LIN {X 0,Y 204.883,Z 502.93,A -85,B 0,C 180,E1 -21530.063,E2 -21530.063} C_VEL
LIN {X 0,Y 207.726,Z 494.964,A -85,B 0,C 180,E1 -21532.899,E2 -21532.899} C_VEL
LIN {X 0,Y 210.33,Z 486.837,A -85,B 0,C 180,E1 -21535.21,E2 -21535.21} C_VEL
LIN {X 0,Y 212.639,Z 478.027,A -85,B 0,C 180,E1 -21537.271,E2 -21537.271} C_VEL
LIN {X 0,Y 215.435,Z 466.867,A -85,B 0,C 180,E1 -21539.299,E2 -21539.299} C_VEL
LIN {X 0,Y 217.848,Z 456.062,A -85,B 0,C 180,E1 -21540.809,E2 -21540.809} C_VEL
LIN {X 0,Y 219.818,Z 444.103,A -85,B 0,C 180,E1 -21542.111,E2 -21542.111} C_VEL
LIN {X 0,Y 221.525,Z 430.516,A -85,B 0,C 180,E1 -21543.135,E2 -21543.135} C_VEL
LIN {X 0,Y 222.579,Z 417.478,A -85,B 0,C 180,E1 -21543.751,E2 -21543.751} C_VEL
LIN {X 0,Y 224.876,Z 365.159,A -85,B 0,C 180,E1 -21545.36,E2 -21545.36} C_VEL
LIN {X 0,Y 218.22,Z 351.727,A -85,B 0,C 180,E1 -21547.162,E2 -21547.162} C_VEL
LIN {X 0,Y 211.105,Z 339.207,A -85,B 0,C 180,E1 -21549.189,E2 -21549.189} C_VEL
LIN {X 0,Y 204.724,Z 329.151,A -85,B 0,C 180,E1 -21551.13,E2 -21551.13} C_VEL
LIN {X 0,Y 202.531,Z 325.685,A -85,B 0,C 180,E1 -21551.84,E2 -21551.84} C_VEL
LIN {X 0,Y 200.323,Z 322.897,A -85,B 0,C 180,E1 -21552.544,E2 -21552.544} C_VEL
LIN {X 0,Y 199.618,Z 320.611,A -85,B 0,C 180,E1 -21552.884,E2 -21552.884} C_VEL
LIN {X 0,Y 199.586,Z 320.596,A -85,B 0,C 180,E1 -21558.006,E2 -21558.006} C_VEL
LIN {X 0,Y 199.617,Z 320.622,A -85,B 0,C 180,E1 -21560.768,E2 -21560.768} C_VEL
LIN {X 0,Y 199.619,Z 320.62,A -85,B 0,C 180,E1 -21565.714,E2 -21565.714} C_VEL
LIN {X 0,Y 199.699,Z 320.598,A -85,B 0,C 180,E1 -21568.137,E2 -21568.137} C_VEL
LIN {X 0,Y 199.782,Z 320.599,A -85,B 0,C 180,E1 -21573.034,E2 -21573.034} C_VEL
LIN {X 0,Y 206.99,Z 349.218,A -85,B 0,C 180,E1 -21575.078,E2 -21575.078} C_VEL
LIN {X 0,Y 203.484,Z 423.442,A -85,B 0,C 180,E1 -21579.706,E2 -21579.706} C_VEL
LIN {X 0,Y 202.574,Z 437.8,A -85,B 0,C 180,E1 -21581.019,E2 -21581.019} C_VEL
LIN {X 0,Y 201.78,Z 450.031,A -85,B 0,C 180,E1 -21582.518,E2 -21582.518} C_VEL
LIN {X 0,Y 201.022,Z 459.956,A -85,B 0,C 180,E1 -21584.019,E2 -21584.019} C_VEL
LIN {X 0,Y 200.03,Z 472.119,A -85,B 0,C 180,E1 -21586.281,E2 -21586.281} C_VEL
LIN {X 0,Y 199.173,Z 483.028,A -85,B 0,C 180,E1 -21588.809,E2 -21588.809} C_VEL
LIN {X 0,Y 198.588,Z 492.082,A -85,B 0,C 180,E1 -21591.349,E2 -21591.349} C_VEL
LIN {X 0,Y 198.092,Z 499.573,A -85,B 0,C 180,E1 -21593.89,E2 -21593.89} C_VEL
LIN {X 0,Y 197.871,Z 507.068,A -85,B 0,C 180,E1 -21596.946,E2 -21596.946} C_VEL
LIN {X 0,Y 197.683,Z 513.047,A -85,B 0,C 180,E1 -21600,E2 -21600} C_VEL
LIN {X 0,Y 197.864,Z 517.861,A -85,B 0,C 180,E1 -21603.054,E2 -21603.054} C_VEL
LIN {X 0,Y 198.329,Z 521.612,A -85,B 0,C 180,E1 -21606.102,E2 -21606.102} C_VEL
LIN {X 0,Y 199.664,Z 525.148,A -85,B 0,C 180,E1 -21610.137,E2 -21610.137} C_VEL
LIN {X 0,Y 202.176,Z 527.196,A -85,B 0,C 180,E1 -21614.083,E2 -21614.083} C_VEL
LIN {X 0,Y 205.529,Z 527.784,A -85,B 0,C 180,E1 -21617.924,E2 -21617.924} C_VEL
LIN {X 0,Y 210.067,Z 526.862,A -85,B 0,C 180,E1 -21621.593,E2 -21621.593} C_VEL
LIN {X 0,Y 215.556,Z 524.507,A -85,B 0,C 180,E1 -21625.078,E2 -21625.078} C_VEL
LIN {X 0,Y 221.972,Z 520.613,A -85,B 0,C 180,E1 -21628.355,E2 -21628.355} C_VEL
LIN {X 0,Y 227.936,Z 516.178,A -85,B 0,C 180,E1 -21630.852,E2 -21630.852} C_VEL
LIN {X 0,Y 230.413,Z 513.934,A -85,B 0,C 180,E1 -21632.07,E2 -21632.07} C_VEL
LIN {X 0,Y 235.965,Z 507.455,A -85,B 0,C 180,E1 -21635.911,E2 -21635.911} C_VEL
LIN {X 0,Y 238.533,Z 504.702,A -85,B 0,C 180,E1 -21636.994,E2 -21636.994} C_VEL
LIN {X 0,Y 239.576,Z 503.651,A -85,B 0,C 180,E1 -21637.301,E2 -21637.301} C_VEL
LIN {X 0,Y 246.733,Z 495.901,A -85,B 0,C 180,E1 -21639.118,E2 -21639.118} C_VEL
LIN {X 0,Y 253.535,Z 487.509,A -85,B 0,C 180,E1 -21640.649,E2 -21640.649} C_VEL
LIN {X 0,Y 260.762,Z 477.305,A -85,B 0,C 180,E1 -21642.1,E2 -21642.1} C_VEL
LIN {X 0,Y 267.508,Z 466.194,A -85,B 0,C 180,E1 -21643.343,E2 -21643.343} C_VEL
LIN {X 0,Y 273.686,Z 454.125,A -85,B 0,C 180,E1 -21644.356,E2 -21644.356} C_VEL
LIN {X 0,Y 273.26,Z 455.121,A -85,B 0,C 180,E1 -21644.754,E2 -21644.754} C_VEL
LIN {X 0,Y 266.867,Z 467.844,A -85,B 0,C 180,E1 -21645.596,E2 -21645.596} C_VEL
LIN {X 0,Y 259.241,Z 480.574,A -85,B 0,C 180,E1 -21646.747,E2 -21646.747} C_VEL
LIN {X 0,Y 253.403,Z 489.105,A -85,B 0,C 180,E1 -21647.733,E2 -21647.733} C_VEL
LIN {X 0,Y 246.637,Z 497.975,A -85,B 0,C 180,E1 -21649.049,E2 -21649.049} C_VEL
LIN {X 0,Y 238.874,Z 507.03,A -85,B 0,C 180,E1 -21650.759,E2 -21650.759} C_VEL
LIN {X 0,Y 230.486,Z 515.708,A -85,B 0,C 180,E1 -21652.969,E2 -21652.969} C_VEL
LIN {X 0,Y 222.797,Z 522.767,A -85,B 0,C 180,E1 -21655.401,E2 -21655.401} C_VEL
LIN {X 0,Y 216.779,Z 527.728,A -85,B 0,C 180,E1 -21657.659,E2 -21657.659} C_VEL
LIN {X 0,Y 209.493,Z 532.953,A -85,B 0,C 180,E1 -21660.891,E2 -21660.891} C_VEL
LIN {X 0,Y 204.769,Z 535.863,A -85,B 0,C 180,E1 -21663.499,E2 -21663.499} C_VEL
LIN {X 0,Y 199.666,Z 538.52,A -85,B 0,C 180,E1 -21667.218,E2 -21667.218} C_VEL
LIN {X 0,Y 195.58,Z 539.845,A -85,B 0,C 180,E1 -21671.129,E2 -21671.129} C_VEL
LIN {X 0,Y 192.79,Z 539.808,A -85,B 0,C 180,E1 -21675.214,E2 -21675.214} C_VEL
LIN {X 0,Y 191.317,Z 538.398,A -85,B 0,C 180,E1 -21679.414,E2 -21679.414} C_VEL
LIN {X 0,Y 191.037,Z 537.758,A -85,B 0,C 180,E1 -21680.869,E2 -21680.869} C_VEL
LIN {X 0,Y 190.528,Z 539.752,A -85,B 0,C 180,E1 -21683.645,E2 -21683.645} C_VEL
LIN {X 0,Y 190.385,Z 540.768,A -85,B 0,C 180,E1 -21685.764,E2 -21685.764} C_VEL
LIN {X 0,Y 190.403,Z 541.392,A -85,B 0,C 180,E1 -21687.883,E2 -21687.883} C_VEL
LIN {X 0,Y 190.598,Z 541.618,A -85,B 0,C 180,E1 -21689.998,E2 -21689.998} C_VEL
LIN {X 0,Y 190.41,Z 541.379,A -85,B 0,C 180,E1 -21692.113,E2 -21692.113} C_VEL
LIN {X 0,Y 190.302,Z 540.701,A -85,B 0,C 180,E1 -21694.341,E2 -21694.341} C_VEL
LIN {X 0,Y 190.306,Z 539.712,A -85,B 0,C 180,E1 -21696.359,E2 -21696.359} C_VEL
LIN {X 0,Y 190.479,Z 538.255,A -85,B 0,C 180,E1 -21698.485,E2 -21698.485} C_VEL
LIN {X 0,Y 191.094,Z 535.243,A -85,B 0,C 180,E1 -21701.668,E2 -21701.668} C_VEL
LIN {X 0,Y 192.189,Z 531.169,A -85,B 0,C 180,E1 -21704.829,E2 -21704.829} C_VEL
LIN {X 0,Y 194.299,Z 524.907,A -85,B 0,C 180,E1 -21708.449,E2 -21708.449} C_VEL
LIN {X 0,Y 196.303,Z 519.321,A -85,B 0,C 180,E1 -21710.976,E2 -21710.976} C_VEL
LIN {X 0,Y 198.955,Z 511.125,A -85,B 0,C 180,E1 -21713.966,E2 -21713.966} C_VEL
LIN {X 0,Y 201.69,Z 502.727,A -85,B 0,C 180,E1 -21716.375,E2 -21716.375} C_VEL
LIN {X 0,Y 204.869,Z 492.34,A -85,B 0,C 180,E1 -21718.701,E2 -21718.701} C_VEL
LIN {X 0,Y 207.651,Z 482.066,A -85,B 0,C 180,E1 -21720.507,E2 -21720.507} C_VEL
LIN {X 0,Y 210.277,Z 470.801,A -85,B 0,C 180,E1 -21722.042,E2 -21722.042} C_VEL
LIN {X 0,Y 212.675,Z 457.931,A -85,B 0,C 180,E1 -21723.322,E2 -21723.322} C_VEL
LIN {X 0,Y 214.527,Z 445.105,A -85,B 0,C 180,E1 -21724.193,E2 -21724.193} C_VEL
LIN {X 0,Y 215.524,Z 431.944,A -85,B 0,C 180,E1 -21724.76,E2 -21724.76} C_VEL
LIN {X 0,Y 217.316,Z 391.03,A -85,B 0,C 180,E1 -21726.05,E2 -21726.05} C_VEL
LIN {X 0,Y 214.641,Z 363.738,A -85,B 0,C 180,E1 -21727.683,E2 -21727.683} C_VEL
LIN {X 0,Y 210.098,Z 349.908,A -85,B 0,C 180,E1 -21729.23,E2 -21729.23} C_VEL
LIN {X 0,Y 204.593,Z 340.582,A -85,B 0,C 180,E1 -21730.911,E2 -21730.911} C_VEL
LIN {X 0,Y 200.055,Z 333.574,A -85,B 0,C 180,E1 -21732.368,E2 -21732.368} C_VEL
LIN {X 0,Y 197.462,Z 329.773,A -85,B 0,C 180,E1 -21733.238,E2 -21733.238} C_VEL
LIN {X 0,Y 195.165,Z 326.199,A -85,B 0,C 180,E1 -21734.048,E2 -21734.048} C_VEL
LIN {X 0,Y 193.201,Z 323.758,A -85,B 0,C 180,E1 -21734.734,E2 -21734.734} C_VEL
LIN {X 0,Y 192.549,Z 321.496,A -85,B 0,C 180,E1 -21735.102,E2 -21735.102} C_VEL
LIN {X 0,Y 192.499,Z 321.494,A -85,B 0,C 180,E1 -21740.054,E2 -21740.054} C_VEL
LIN {X 0,Y 192.551,Z 321.489,A -85,B 0,C 180,E1 -21744.268,E2 -21744.268} C_VEL
LIN {X 0,Y 192.598,Z 321.492,A -85,B 0,C 180,E1 -21747.06,E2 -21747.06} C_VEL
LIN {X 0,Y 192.612,Z 321.493,A -85,B 0,C 180,E1 -21751.683,E2 -21751.683} C_VEL
LIN {X 0,Y 192.655,Z 321.486,A -85,B 0,C 180,E1 -21756.342,E2 -21756.342} C_VEL
LIN {X 0,Y 192.687,Z 321.438,A -85,B 0,C 180,E1 -21761.491,E2 -21761.491} C_VEL
LIN {X 0,Y 192.731,Z 321.453,A -85,B 0,C 180,E1 -21765.211,E2 -21765.211} C_VEL
LIN {X 0,Y 192.938,Z 321.445,A -85,B 0,C 180,E1 -21769.566,E2 -21769.566} C_VEL
LIN {X 0,Y 192.956,Z 321.393,A -85,B 0,C 180,E1 -21773.727,E2 -21773.727} C_VEL
LIN {X 0,Y 193.222,Z 321.399,A -85,B 0,C 180,E1 -21777.916,E2 -21777.916} C_VEL
LIN {X 0,Y 193.404,Z 321.391,A -85,B 0,C 180,E1 -21780,E2 -21780} C_VEL
LIN {X 0,Y 192.924,Z 321.441,A -85,B 0,C 180,E1 -21784.178,E2 -21784.178} C_VEL
LIN {X 0,Y 193.016,Z 321.434,A -85,B 0,C 180,E1 -21788.375,E2 -21788.375} C_VEL
LIN {X 0,Y 192.784,Z 321.471,A -85,B 0,C 180,E1 -21792.635,E2 -21792.635} C_VEL
LIN {X 0,Y 192.712,Z 321.454,A -85,B 0,C 180,E1 -21796.963,E2 -21796.963} C_VEL
LIN {X 0,Y 192.602,Z 321.493,A -85,B 0,C 180,E1 -21801.401,E2 -21801.401} C_VEL
LIN {X 0,Y 192.633,Z 321.47,A -85,B 0,C 180,E1 -21804.209,E2 -21804.209} C_VEL
LIN {X 0,Y 192.596,Z 321.495,A -85,B 0,C 180,E1 -21808.867,E2 -21808.867} C_VEL
LIN {X 0,Y 192.589,Z 321.482,A -85,B 0,C 180,E1 -21813.188,E2 -21813.188} C_VEL
LIN {X 0,Y 192.545,Z 321.485,A -85,B 0,C 180,E1 -21818.354,E2 -21818.354} C_VEL
LIN {X 0,Y 192.484,Z 321.496,A -85,B 0,C 180,E1 -21823.097,E2 -21823.097} C_VEL
LIN {X 0,Y 192.549,Z 321.515,A -85,B 0,C 180,E1 -21825.4,E2 -21825.4} C_VEL
LIN {X 0,Y 193.375,Z 324.086,A -85,B 0,C 180,E1 -21825.774,E2 -21825.774} C_VEL
LIN {X 0,Y 195.707,Z 326.993,A -85,B 0,C 180,E1 -21826.585,E2 -21826.585} C_VEL
LIN {X 0,Y 197.792,Z 330.187,A -85,B 0,C 180,E1 -21827.314,E2 -21827.314} C_VEL
LIN {X 0,Y 203.771,Z 339.212,A -85,B 0,C 180,E1 -21829.272,E2 -21829.272} C_VEL
LIN {X 0,Y 210.873,Z 351.252,A -85,B 0,C 180,E1 -21831.445,E2 -21831.445} C_VEL
LIN {X 0,Y 217.687,Z 364.631,A -85,B 0,C 180,E1 -21833.415,E2 -21833.415} C_VEL
LIN {X 0,Y 218.98,Z 367.37,A -85,B 0,C 180,E1 -21833.778,E2 -21833.778} C_VEL
LIN {X 0,Y 216.238,Z 422.514,A -85,B 0,C 180,E1 -21835.528,E2 -21835.528} C_VEL
LIN {X 0,Y 215.03,Z 435.02,A -85,B 0,C 180,E1 -21836.249,E2 -21836.249} C_VEL
LIN {X 0,Y 213.234,Z 447.586,A -85,B 0,C 180,E1 -21837.339,E2 -21837.339} C_VEL
LIN {X 0,Y 211.136,Z 458.838,A -85,B 0,C 180,E1 -21838.663,E2 -21838.663} C_VEL
LIN {X 0,Y 208.673,Z 469.175,A -85,B 0,C 180,E1 -21840.216,E2 -21840.216} C_VEL
LIN {X 0,Y 206.125,Z 478.927,A -85,B 0,C 180,E1 -21842.1,E2 -21842.1} C_VEL
LIN {X 0,Y 203.422,Z 488.432,A -85,B 0,C 180,E1 -21844.43,E2 -21844.43} C_VEL
LIN {X 0,Y 200.224,Z 497.77,A -85,B 0,C 180,E1 -21847.29,E2 -21847.29} C_VEL
LIN {X 0,Y 197.517,Z 505.216,A -85,B 0,C 180,E1 -21850.246,E2 -21850.246} C_VEL
LIN {X 0,Y 195.288,Z 511.189,A -85,B 0,C 180,E1 -21853.27,E2 -21853.27} C_VEL
LIN {X 0,Y 193.48,Z 515.906,A -85,B 0,C 180,E1 -21856.345,E2 -21856.345} C_VEL
LIN {X 0,Y 192.195,Z 519.505,A -85,B 0,C 180,E1 -21859.467,E2 -21859.467} C_VEL
LIN {X 0,Y 191.243,Z 522.257,A -85,B 0,C 180,E1 -21862.852,E2 -21862.852} C_VEL
LIN {X 0,Y 190.77,Z 523.755,A -85,B 0,C 180,E1 -21865.777,E2 -21865.777} C_VEL
LIN {X 0,Y 190.523,Z 524.593,A -85,B 0,C 180,E1 -21870.002,E2 -21870.002} C_VEL
LIN {X 0,Y 190.573,Z 524.396,A -85,B 0,C 180,E1 -21872.116,E2 -21872.116} C_VEL
LIN {X 0,Y 190.77,Z 523.809,A -85,B 0,C 180,E1 -21874.228,E2 -21874.228} C_VEL
LIN {X 0,Y 191.565,Z 521.476,A -85,B 0,C 180,E1 -21878.441,E2 -21878.441} C_VEL
LIN {X 0,Y 192.512,Z 518.607,A -85,B 0,C 180,E1 -21881.585,E2 -21881.585} C_VEL
LIN {X 0,Y 193.961,Z 514.699,A -85,B 0,C 180,E1 -21884.695,E2 -21884.695} C_VEL
LIN {X 0,Y 195.918,Z 509.63,A -85,B 0,C 180,E1 -21887.755,E2 -21887.755} C_VEL
LIN {X 0,Y 198.239,Z 503.242,A -85,B 0,C 180,E1 -21890.766,E2 -21890.766} C_VEL
LIN {X 0,Y 201.218,Z 495.274,A -85,B 0,C 180,E1 -21893.684,E2 -21893.684} C_VEL
LIN {X 0,Y 203.728,Z 487.809,A -85,B 0,C 180,E1 -21895.877,E2 -21895.877} C_VEL
LIN {X 0,Y 206.372,Z 478.331,A -85,B 0,C 180,E1 -21898.172,E2 -21898.172} C_VEL
LIN {X 0,Y 209.302,Z 467.166,A -85,B 0,C 180,E1 -21900.245,E2 -21900.245} C_VEL
LIN {X 0,Y 211.792,Z 456.355,A -85,B 0,C 180,E1 -21901.791,E2 -21901.791} C_VEL
LIN {X 0,Y 213.84,Z 444.384,A -85,B 0,C 180,E1 -21903.122,E2 -21903.122} C_VEL
LIN {X 0,Y 215.604,Z 431.091,A -85,B 0,C 180,E1 -21904.142,E2 -21904.142} C_VEL
LIN {X 0,Y 216.702,Z 418.103,A -85,B 0,C 180,E1 -21904.776,E2 -21904.776} C_VEL
LIN {X 0,Y 219.02,Z 367.335,A -85,B 0,C 180,E1 -21906.374,E2 -21906.374} C_VEL
LIN {X 0,Y 212.213,Z 353.671,A -85,B 0,C 180,E1 -21908.327,E2 -21908.327} C_VEL
LIN {X 0,Y 205.194,Z 341.395,A -85,B 0,C 180,E1 -21910.458,E2 -21910.458} C_VEL
LIN {X 0,Y 197.936,Z 330.286,A -85,B 0,C 180,E1 -21912.825,E2 -21912.825} C_VEL
LIN {X 0,Y 195.708,Z 326.922,A -85,B 0,C 180,E1 -21913.604,E2 -21913.604} C_VEL
LIN {X 0,Y 194.407,Z 325.394,A -85,B 0,C 180,E1 -21914.05,E2 -21914.05} C_VEL
LIN {X 0,Y 192.884,Z 322.876,A -85,B 0,C 180,E1 -21914.621,E2 -21914.621} C_VEL
LIN {X 0,Y 192.56,Z 321.457,A -85,B 0,C 180,E1 -21914.841,E2 -21914.841} C_VEL
LIN {X 0,Y 192.525,Z 321.505,A -85,B 0,C 180,E1 -21920.052,E2 -21920.052} C_VEL
LIN {X 0,Y 192.566,Z 321.487,A -85,B 0,C 180,E1 -21924.271,E2 -21924.271} C_VEL
LIN {X 0,Y 192.614,Z 321.489,A -85,B 0,C 180,E1 -21927.06,E2 -21927.06} C_VEL
LIN {X 0,Y 192.736,Z 321.478,A -85,B 0,C 180,E1 -21932.832,E2 -21932.832} C_VEL
LIN {X 0,Y 199.89,Z 350.039,A -85,B 0,C 180,E1 -21934.932,E2 -21934.932} C_VEL
LIN {X 0,Y 196.37,Z 424.117,A -85,B 0,C 180,E1 -21939.782,E2 -21939.782} C_VEL
LIN {X 0,Y 195.447,Z 438.02,A -85,B 0,C 180,E1 -21941.117,E2 -21941.117} C_VEL
LIN {X 0,Y 194.654,Z 450.194,A -85,B 0,C 180,E1 -21942.67,E2 -21942.67} C_VEL
LIN {X 0,Y 193.87,Z 460.065,A -85,B 0,C 180,E1 -21944.224,E2 -21944.224} C_VEL
LIN {X 0,Y 192.912,Z 472.254,A -85,B 0,C 180,E1 -21946.57,E2 -21946.57} C_VEL
LIN {X 0,Y 192.147,Z 482.17,A -85,B 0,C 180,E1 -21948.929,E2 -21948.929} C_VEL
LIN {X 0,Y 191.55,Z 491.348,A -85,B 0,C 180,E1 -21951.561,E2 -21951.561} C_VEL
LIN {X 0,Y 191.037,Z 499.514,A -85,B 0,C 180,E1 -21954.393,E2 -21954.393} C_VEL
LIN {X 0,Y 190.874,Z 506.603,A -85,B 0,C 180,E1 -21957.362,E2 -21957.362} C_VEL
LIN {X 0,Y 190.701,Z 513.621,A -85,B 0,C 180,E1 -21961.056,E2 -21961.056} C_VEL
LIN {X 0,Y 190.993,Z 518.377,A -85,B 0,C 180,E1 -21964.22,E2 -21964.22} C_VEL
LIN {X 0,Y 191.885,Z 523.194,A -85,B 0,C 180,E1 -21968.532,E2 -21968.532} C_VEL
LIN {X 0,Y 193.882,Z 526.29,A -85,B 0,C 180,E1 -21972.562,E2 -21972.562} C_VEL
LIN {X 0,Y 196.955,Z 527.964,A -85,B 0,C 180,E1 -21976.587,E2 -21976.587} C_VEL
LIN {X 0,Y 201.058,Z 528.212,A -85,B 0,C 180,E1 -21980.46,E2 -21980.46} C_VEL
LIN {X 0,Y 206.273,Z 527.053,A -85,B 0,C 180,E1 -21984.133,E2 -21984.133} C_VEL
LIN {X 0,Y 212.548,Z 524.388,A -85,B 0,C 180,E1 -21987.575,E2 -21987.575} C_VEL
LIN {X 0,Y 217.803,Z 521.431,A -85,B 0,C 180,E1 -21990.01,E2 -21990.01} C_VEL
LIN {X 0,Y 225.621,Z 515.995,A -85,B 0,C 180,E1 -21993.033,E2 -21993.033} C_VEL
LIN {X 0,Y 232.035,Z 510.749,A -85,B 0,C 180,E1 -21995.133,E2 -21995.133} C_VEL
LIN {X 0,Y 239.576,Z 503.651,A -85,B 0,C 180,E1 -21997.301,E2 -21997.301} C_VEL
LIN {X 0,Y 242.542,Z 500.561,A -85,B 0,C 180,E1 -21998.271,E2 -21998.271} C_VEL
LIN {X 0,Y 249.703,Z 491.757,A -85,B 0,C 180,E1 -22001.466,E2 -22001.466} C_VEL
LIN {X 0,Y 252.5,Z 488.196,A -85,B 0,C 180,E1 -22002.314,E2 -22002.314} C_VEL
LIN {X 0,Y 253.549,Z 486.877,A -85,B 0,C 180,E1 -22002.537,E2 -22002.537} C_VEL
LIN {X 0,Y 261.752,Z 475.604,A -85,B 0,C 180,E1 -22004.007,E2 -22004.007} C_VEL
LIN {X 0,Y 262.445,Z 474.552,A -85,B 0,C 180,E1 -22004.127,E2 -22004.127} C_VEL
LIN {X 0,Y 263.075,Z 473.63,A -85,B 0,C 180,E1 -22004.474,E2 -22004.474} C_VEL
LIN {X 0,Y 254.249,Z 486.612,A -85,B 0,C 180,E1 -22005.734,E2 -22005.734} C_VEL
LIN {X 0,Y 245.683,Z 497.363,A -85,B 0,C 180,E1 -22007.202,E2 -22007.202} C_VEL
LIN {X 0,Y 236.249,Z 507.695,A -85,B 0,C 180,E1 -22009.119,E2 -22009.119} C_VEL
LIN {X 0,Y 227.457,Z 516.071,A -85,B 0,C 180,E1 -22011.265,E2 -22011.265} C_VEL
LIN {X 0,Y 219.329,Z 522.916,A -85,B 0,C 180,E1 -22013.642,E2 -22013.642} C_VEL
LIN {X 0,Y 212.921,Z 527.704,A -85,B 0,C 180,E1 -22015.864,E2 -22015.864} C_VEL
LIN {X 0,Y 205.155,Z 532.761,A -85,B 0,C 180,E1 -22019.077,E2 -22019.077} C_VEL
LIN {X 0,Y 198.463,Z 536.325,A -85,B 0,C 180,E1 -22022.588,E2 -22022.588} C_VEL
LIN {X 0,Y 193.144,Z 538.52,A -85,B 0,C 180,E1 -22026.403,E2 -22026.403} C_VEL
LIN {X 0,Y 188.879,Z 539.414,A -85,B 0,C 180,E1 -22030.433,E2 -22030.433} C_VEL
LIN {X 0,Y 185.963,Z 539.002,A -85,B 0,C 180,E1 -22034.658,E2 -22034.658} C_VEL
LIN {X 0,Y 184.399,Z 537.272,A -85,B 0,C 180,E1 -22039.012,E2 -22039.012} C_VEL
LIN {X 0,Y 184.242,Z 536.881,A -85,B 0,C 180,E1 -22039.836,E2 -22039.836} C_VEL
LIN {X 0,Y 183.454,Z 539.434,A -85,B 0,C 180,E1 -22043.398,E2 -22043.398} C_VEL
LIN {X 0,Y 183.309,Z 540.451,A -85,B 0,C 180,E1 -22045.6,E2 -22045.6} C_VEL
LIN {X 0,Y 183.305,Z 541.074,A -85,B 0,C 180,E1 -22047.801,E2 -22047.801} C_VEL
LIN {X 0,Y 183.507,Z 541.302,A -85,B 0,C 180,E1 -22049.998,E2 -22049.998} C_VEL
LIN {X 0,Y 183.214,Z 540.509,A -85,B 0,C 180,E1 -22054.172,E2 -22054.172} C_VEL
LIN {X 0,Y 183.225,Z 539.393,A -85,B 0,C 180,E1 -22056.605,E2 -22056.605} C_VEL
LIN {X 0,Y 183.421,Z 537.935,A -85,B 0,C 180,E1 -22058.814,E2 -22058.814} C_VEL
LIN {X 0,Y 184.109,Z 534.924,A -85,B 0,C 180,E1 -22062.117,E2 -22062.117} C_VEL
LIN {X 0,Y 185.311,Z 530.851,A -85,B 0,C 180,E1 -22065.393,E2 -22065.393} C_VEL
LIN {X 0,Y 187.535,Z 524.589,A -85,B 0,C 180,E1 -22069.14,E2 -22069.14} C_VEL
LIN {X 0,Y 189.836,Z 518.278,A -85,B 0,C 180,E1 -22072.062,E2 -22072.062} C_VEL
LIN {X 0,Y 192.436,Z 510.807,A -85,B 0,C 180,E1 -22074.832,E2 -22074.832} C_VEL
LIN {X 0,Y 195.346,Z 502.413,A -85,B 0,C 180,E1 -22077.301,E2 -22077.301} C_VEL
LIN {X 0,Y 198.662,Z 492.029,A -85,B 0,C 180,E1 -22079.685,E2 -22079.685} C_VEL
LIN {X 0,Y 201.933,Z 480.342,A -85,B 0,C 180,E1 -22081.76,E2 -22081.76} C_VEL
LIN {X 0,Y 204.713,Z 468.568,A -85,B 0,C 180,E1 -22083.316,E2 -22083.316} C_VEL
LIN {X 0,Y 207.009,Z 456.373,A -85,B 0,C 180,E1 -22084.507,E2 -22084.507} C_VEL
LIN {X 0,Y 208.863,Z 443.224,A -85,B 0,C 180,E1 -22085.375,E2 -22085.375} C_VEL
LIN {X 0,Y 209.912,Z 428.171,A -85,B 0,C 180,E1 -22085.978,E2 -22085.978} C_VEL
LIN {X 0,Y 211.578,Z 392.104,A -85,B 0,C 180,E1 -22087.135,E2 -22087.135} C_VEL
LIN {X 0,Y 209.174,Z 366.126,A -85,B 0,C 180,E1 -22088.737,E2 -22088.737} C_VEL
LIN {X 0,Y 205.147,Z 353.764,A -85,B 0,C 180,E1 -22090.187,E2 -22090.187} C_VEL
LIN {X 0,Y 200.121,Z 345.122,A -85,B 0,C 180,E1 -22091.808,E2 -22091.808} C_VEL
LIN {X 0,Y 193.96,Z 335.536,A -85,B 0,C 180,E1 -22093.922,E2 -22093.922} C_VEL
LIN {X 0,Y 190.873,Z 331.133,A -85,B 0,C 180,E1 -22095.042,E2 -22095.042} C_VEL
LIN {X 0,Y 188.698,Z 327.695,A -85,B 0,C 180,E1 -22095.885,E2 -22095.885} C_VEL
LIN {X 0,Y 186.337,Z 325.039,A -85,B 0,C 180,E1 -22096.778,E2 -22096.778} C_VEL
LIN {X 0,Y 185.429,Z 322.374,A -85,B 0,C 180,E1 -22097.258,E2 -22097.258} C_VEL
LIN {X 0,Y 185.494,Z 322.375,A -85,B 0,C 180,E1 -22102.712,E2 -22102.712} C_VEL
LIN {X 0,Y 185.524,Z 322.372,A -85,B 0,C 180,E1 -22107.971,E2 -22107.971} C_VEL
LIN {X 0,Y 185.54,Z 322.367,A -85,B 0,C 180,E1 -22110.594,E2 -22110.594} C_VEL
LIN {X 0,Y 185.555,Z 322.362,A -85,B 0,C 180,E1 -22115.378,E2 -22115.378} C_VEL
LIN {X 0,Y 185.618,Z 322.319,A -85,B 0,C 180,E1 -22121.178,E2 -22121.178} C_VEL
LIN {X 0,Y 185.66,Z 322.321,A -85,B 0,C 180,E1 -22124.634,E2 -22124.634} C_VEL
LIN {X 0,Y 185.88,Z 322.325,A -85,B 0,C 180,E1 -22129.419,E2 -22129.419} C_VEL
LIN {X 0,Y 185.921,Z 322.269,A -85,B 0,C 180,E1 -22133.489,E2 -22133.489} C_VEL
LIN {X 0,Y 186.168,Z 322.275,A -85,B 0,C 180,E1 -22137.837,E2 -22137.837} C_VEL
LIN {X 0,Y 186.37,Z 322.267,A -85,B 0,C 180,E1 -22140,E2 -22140} C_VEL
LIN {X 0,Y 185.872,Z 322.32,A -85,B 0,C 180,E1 -22144.337,E2 -22144.337} C_VEL
LIN {X 0,Y 185.966,Z 322.309,A -85,B 0,C 180,E1 -22148.695,E2 -22148.695} C_VEL
LIN {X 0,Y 185.71,Z 322.352,A -85,B 0,C 180,E1 -22153.124,E2 -22153.124} C_VEL
LIN {X 0,Y 185.649,Z 322.334,A -85,B 0,C 180,E1 -22157.629,E2 -22157.629} C_VEL
LIN {X 0,Y 185.565,Z 322.366,A -85,B 0,C 180,E1 -22162.256,E2 -22162.256} C_VEL
LIN {X 0,Y 185.571,Z 322.347,A -85,B 0,C 180,E1 -22164.647,E2 -22164.647} C_VEL
LIN {X 0,Y 185.538,Z 322.372,A -85,B 0,C 180,E1 -22169.501,E2 -22169.501} C_VEL
LIN {X 0,Y 185.492,Z 322.378,A -85,B 0,C 180,E1 -22174.634,E2 -22174.634} C_VEL
LIN {X 0,Y 185.499,Z 322.363,A -85,B 0,C 180,E1 -22177.315,E2 -22177.315} C_VEL
LIN {X 0,Y 185.465,Z 322.383,A -85,B 0,C 180,E1 -22180.726,E2 -22180.726} C_VEL
LIN {X 0,Y 185.448,Z 322.372,A -85,B 0,C 180,E1 -22183.2,E2 -22183.2} C_VEL
LIN {X 0,Y 186.506,Z 325.331,A -85,B 0,C 180,E1 -22183.734,E2 -22183.734} C_VEL
LIN {X 0,Y 188.784,Z 327.935,A -85,B 0,C 180,E1 -22184.596,E2 -22184.596} C_VEL
LIN {X 0,Y 191.043,Z 331.325,A -85,B 0,C 180,E1 -22185.461,E2 -22185.461} C_VEL
LIN {X 0,Y 197.255,Z 340.534,A -85,B 0,C 180,E1 -22187.673,E2 -22187.673} C_VEL
LIN {X 0,Y 203.62,Z 350.983,A -85,B 0,C 180,E1 -22189.773,E2 -22189.773} C_VEL
LIN {X 0,Y 211.367,Z 365.682,A -85,B 0,C 180,E1 -22192.167,E2 -22192.167} C_VEL
LIN {X 0,Y 213.149,Z 369.458,A -85,B 0,C 180,E1 -22192.698,E2 -22192.698} C_VEL
LIN {X 0,Y 210.402,Z 423.022,A -85,B 0,C 180,E1 -22194.443,E2 -22194.443} C_VEL
LIN {X 0,Y 209.087,Z 436.025,A -85,B 0,C 180,E1 -22195.227,E2 -22195.227} C_VEL
LIN {X 0,Y 207.123,Z 448.965,A -85,B 0,C 180,E1 -22196.395,E2 -22196.395} C_VEL
LIN {X 0,Y 204.78,Z 460.784,A -85,B 0,C 180,E1 -22197.865,E2 -22197.865} C_VEL
LIN {X 0,Y 201.9,Z 472.015,A -85,B 0,C 180,E1 -22199.689,E2 -22199.689} C_VEL
LIN {X 0,Y 199.229,Z 481.524,A -85,B 0,C 180,E1 -22201.678,E2 -22201.678} C_VEL
LIN {X 0,Y 196.454,Z 490.591,A -85,B 0,C 180,E1 -22204.061,E2 -22204.061} C_VEL
LIN {X 0,Y 193.183,Z 499.42,A -85,B 0,C 180,E1 -22206.98,E2 -22206.98} C_VEL
LIN {X 0,Y 190.452,Z 506.622,A -85,B 0,C 180,E1 -22210.044,E2 -22210.044} C_VEL
LIN {X 0,Y 187.798,Z 513.225,A -85,B 0,C 180,E1 -22213.702,E2 -22213.702} C_VEL
LIN {X 0,Y 186.079,Z 517.551,A -85,B 0,C 180,E1 -22216.905,E2 -22216.905} C_VEL
LIN {X 0,Y 185.215,Z 519.823,A -85,B 0,C 180,E1 -22219.066,E2 -22219.066} C_VEL
LIN {X 0,Y 184.128,Z 522.804,A -85,B 0,C 180,E1 -22222.932,E2 -22222.932} C_VEL
LIN {X 0,Y 183.69,Z 524.072,A -85,B 0,C 180,E1 -22225.614,E2 -22225.614} C_VEL
LIN {X 0,Y 183.498,Z 524.68,A -85,B 0,C 180,E1 -22227.807,E2 -22227.807} C_VEL
LIN {X 0,Y 183.441,Z 524.909,A -85,B 0,C 180,E1 -22230.002,E2 -22230.002} C_VEL
LIN {X 0,Y 183.498,Z 524.712,A -85,B 0,C 180,E1 -22232.197,E2 -22232.197} C_VEL
LIN {X 0,Y 183.69,Z 524.126,A -85,B 0,C 180,E1 -22234.391,E2 -22234.391} C_VEL
LIN {X 0,Y 184.13,Z 522.9,A -85,B 0,C 180,E1 -22237.072,E2 -22237.072} C_VEL
LIN {X 0,Y 185.165,Z 519.967,A -85,B 0,C 180,E1 -22240.942,E2 -22240.942} C_VEL
LIN {X 0,Y 186.534,Z 516.415,A -85,B 0,C 180,E1 -22244.178,E2 -22244.178} C_VEL
LIN {X 0,Y 188.408,Z 511.751,A -85,B 0,C 180,E1 -22247.365,E2 -22247.365} C_VEL
LIN {X 0,Y 190.777,Z 505.836,A -85,B 0,C 180,E1 -22250.488,E2 -22250.488} C_VEL
LIN {X 0,Y 193.666,Z 498.461,A -85,B 0,C 180,E1 -22253.529,E2 -22253.529} C_VEL
LIN {X 0,Y 196.875,Z 489.708,A -85,B 0,C 180,E1 -22256.325,E2 -22256.325} C_VEL
LIN {X 0,Y 199.784,Z 479.793,A -85,B 0,C 180,E1 -22258.872,E2 -22258.872} C_VEL
LIN {X 0,Y 202.855,Z 468.845,A -85,B 0,C 180,E1 -22261.023,E2 -22261.023} C_VEL
LIN {X 0,Y 205.806,Z 456.648,A -85,B 0,C 180,E1 -22262.83,E2 -22262.83} C_VEL
LIN {X 0,Y 207.934,Z 444.665,A -85,B 0,C 180,E1 -22264.19,E2 -22264.19} C_VEL
LIN {X 0,Y 209.744,Z 431.677,A -85,B 0,C 180,E1 -22265.207,E2 -22265.207} C_VEL
LIN {X 0,Y 210.894,Z 418.856,A -85,B 0,C 180,E1 -22265.851,E2 -22265.851} C_VEL
LIN {X 0,Y 213.243,Z 369.52,A -85,B 0,C 180,E1 -22267.443,E2 -22267.443} C_VEL
LIN {X 0,Y 206.109,Z 355.341,A -85,B 0,C 180,E1 -22269.616,E2 -22269.616} C_VEL
LIN {X 0,Y 198.95,Z 343.064,A -85,B 0,C 180,E1 -22271.94,E2 -22271.94} C_VEL
LIN {X 0,Y 193.496,Z 334.902,A -85,B 0,C 180,E1 -22273.829,E2 -22273.829} C_VEL
LIN {X 0,Y 190.897,Z 331.07,A -85,B 0,C 180,E1 -22274.787,E2 -22274.787} C_VEL
LIN {X 0,Y 188.783,Z 327.737,A -85,B 0,C 180,E1 -22275.61,E2 -22275.61} C_VEL
LIN {X 0,Y 186.295,Z 324.87,A -85,B 0,C 180,E1 -22276.56,E2 -22276.56} C_VEL
LIN {X 0,Y 185.486,Z 322.337,A -85,B 0,C 180,E1 -22276.998,E2 -22276.998} C_VEL
LIN {X 0,Y 185.475,Z 322.38,A -85,B 0,C 180,E1 -22279.897,E2 -22279.897} C_VEL
LIN {X 0,Y 185.512,Z 322.363,A -85,B 0,C 180,E1 -22282.712,E2 -22282.712} C_VEL
LIN {X 0,Y 185.549,Z 322.36,A -85,B 0,C 180,E1 -22287.976,E2 -22287.976} C_VEL
LIN {X 0,Y 185.731,Z 322.521,A -85,B 0,C 180,E1 -22292.66,E2 -22292.66} C_VEL
LIN {X 0,Y 192.824,Z 350.429,A -85,B 0,C 180,E1 -22294.776,E2 -22294.776} C_VEL
LIN {X 0,Y 189.275,Z 424.941,A -85,B 0,C 180,E1 -22299.912,E2 -22299.912} C_VEL
LIN {X 0,Y 188.289,Z 439.198,A -85,B 0,C 180,E1 -22301.361,E2 -22301.361} C_VEL
LIN {X 0,Y 187.339,Z 453.762,A -85,B 0,C 180,E1 -22303.378,E2 -22303.378} C_VEL
LIN {X 0,Y 186.235,Z 467.143,A -85,B 0,C 180,E1 -22305.801,E2 -22305.801} C_VEL
LIN {X 0,Y 185.405,Z 478.02,A -85,B 0,C 180,E1 -22308.244,E2 -22308.244} C_VEL
LIN {X 0,Y 184.656,Z 488.781,A -85,B 0,C 180,E1 -22311.243,E2 -22311.243} C_VEL
LIN {X 0,Y 184.075,Z 498.17,A -85,B 0,C 180,E1 -22314.457,E2 -22314.457} C_VEL
LIN {X 0,Y 183.858,Z 506.053,A -85,B 0,C 180,E1 -22317.809,E2 -22317.809} C_VEL
LIN {X 0,Y 183.727,Z 512.305,A -85,B 0,C 180,E1 -22321.096,E2 -22321.096} C_VEL
LIN {X 0,Y 184.01,Z 517.365,A -85,B 0,C 180,E1 -22324.381,E2 -22324.381} C_VEL
LIN {X 0,Y 184.867,Z 522.514,A -85,B 0,C 180,E1 -22328.747,E2 -22328.747} C_VEL
LIN {X 0,Y 186.981,Z 526.054,A -85,B 0,C 180,E1 -22333.033,E2 -22333.033} C_VEL
LIN {X 0,Y 190.166,Z 528.143,A -85,B 0,C 180,E1 -22337.197,E2 -22337.197} C_VEL
LIN {X 0,Y 194.451,Z 528.839,A -85,B 0,C 180,E1 -22341.188,E2 -22341.188} C_VEL
LIN {X 0,Y 199.908,Z 528.093,A -85,B 0,C 180,E1 -22344.953,E2 -22344.953} C_VEL
LIN {X 0,Y 206.423,Z 525.919,A -85,B 0,C 180,E1 -22348.467,E2 -22348.467} C_VEL
LIN {X 0,Y 211.878,Z 523.35,A -85,B 0,C 180,E1 -22350.94,E2 -22350.94} C_VEL
LIN {X 0,Y 220.006,Z 518.524,A -85,B 0,C 180,E1 -22353.989,E2 -22353.989} C_VEL
LIN {X 0,Y 226.642,Z 513.777,A -85,B 0,C 180,E1 -22356.099,E2 -22356.099} C_VEL
LIN {X 0,Y 234.732,Z 507.052,A -85,B 0,C 180,E1 -22358.355,E2 -22358.355} C_VEL
LIN {X 0,Y 243.577,Z 498.387,A -85,B 0,C 180,E1 -22360.481,E2 -22360.481} C_VEL
LIN {X 0,Y 251.454,Z 489.499,A -85,B 0,C 180,E1 -22362.128,E2 -22362.128} C_VEL
LIN {X 0,Y 253.549,Z 486.877,A -85,B 0,C 180,E1 -22362.537,E2 -22362.537} C_VEL
LIN {X 0,Y 253.935,Z 486.393,A -85,B 0,C 180,E1 -22362.812,E2 -22362.812} C_VEL
LIN {X 0,Y 253.506,Z 486.939,A -85,B 0,C 180,E1 -22363.38,E2 -22363.38} C_VEL
LIN {X 0,Y 251.558,Z 489.393,A -85,B 0,C 180,E1 -22364.163,E2 -22364.163} C_VEL
LIN {X 0,Y 249.658,Z 491.694,A -85,B 0,C 180,E1 -22364.635,E2 -22364.635} C_VEL
LIN {X 0,Y 239.887,Z 502.576,A -85,B 0,C 180,E1 -22366.322,E2 -22366.322} C_VEL
LIN {X 0,Y 236.506,Z 505.928,A -85,B 0,C 180,E1 -22366.938,E2 -22366.938} C_VEL
LIN {X 0,Y 228.563,Z 513.269,A -85,B 0,C 180,E1 -22368.615,E2 -22368.615} C_VEL
LIN {X 0,Y 220.901,Z 519.554,A -85,B 0,C 180,E1 -22370.481,E2 -22370.481} C_VEL
LIN {X 0,Y 213.784,Z 524.778,A -85,B 0,C 180,E1 -22372.54,E2 -22372.54} C_VEL
LIN {X 0,Y 205.114,Z 530.37,A -85,B 0,C 180,E1 -22375.571,E2 -22375.571} C_VEL
LIN {X 0,Y 199.135,Z 533.572,A -85,B 0,C 180,E1 -22378.034,E2 -22378.034} C_VEL
LIN {X 0,Y 192.195,Z 536.659,A -85,B 0,C 180,E1 -22381.614,E2 -22381.614} C_VEL
LIN {X 0,Y 186.668,Z 538.417,A -85,B 0,C 180,E1 -22385.532,E2 -22385.532} C_VEL
LIN {X 0,Y 182.21,Z 538.883,A -85,B 0,C 180,E1 -22389.685,E2 -22389.685} C_VEL
LIN {X 0,Y 179.155,Z 538.073,A -85,B 0,C 180,E1 -22394.06,E2 -22394.06} C_VEL
LIN {X 0,Y 177.493,Z 535.931,A -85,B 0,C 180,E1 -22398.724,E2 -22398.724} C_VEL
LIN {X 0,Y 176.827,Z 537.686,A -85,B 0,C 180,E1 -22400.85,E2 -22400.85} C_VEL
LIN {X 0,Y 176.403,Z 539.118,A -85,B 0,C 180,E1 -22403.133,E2 -22403.133} C_VEL
LIN {X 0,Y 176.221,Z 540.196,A -85,B 0,C 180,E1 -22405.595,E2 -22405.595} C_VEL
LIN {X 0,Y 176.417,Z 540.985,A -85,B 0,C 180,E1 -22409.998,E2 -22409.998} C_VEL
LIN {X 0,Y 176.13,Z 540.312,A -85,B 0,C 180,E1 -22414.003,E2 -22414.003} C_VEL
LIN {X 0,Y 176.142,Z 539.075,A -85,B 0,C 180,E1 -22416.872,E2 -22416.872} C_VEL
LIN {X 0,Y 176.385,Z 537.617,A -85,B 0,C 180,E1 -22419.168,E2 -22419.168} C_VEL
LIN {X 0,Y 177.119,Z 534.604,A -85,B 0,C 180,E1 -22422.603,E2 -22422.603} C_VEL
LIN {X 0,Y 178.46,Z 530.533,A -85,B 0,C 180,E1 -22425.999,E2 -22425.999} C_VEL
LIN {X 0,Y 180.816,Z 524.271,A -85,B 0,C 180,E1 -22429.88,E2 -22429.88} C_VEL
LIN {X 0,Y 182.959,Z 518.681,A -85,B 0,C 180,E1 -22432.587,E2 -22432.587} C_VEL
LIN {X 0,Y 185.992,Z 510.491,A -85,B 0,C 180,E1 -22435.754,E2 -22435.754} C_VEL
LIN {X 0,Y 189.046,Z 502.099,A -85,B 0,C 180,E1 -22438.291,E2 -22438.291} C_VEL
LIN {X 0,Y 192.518,Z 491.717,A -85,B 0,C 180,E1 -22440.733,E2 -22440.733} C_VEL
LIN {X 0,Y 195.92,Z 480.033,A -85,B 0,C 180,E1 -22442.855,E2 -22442.855} C_VEL
LIN {X 0,Y 198.822,Z 468.267,A -85,B 0,C 180,E1 -22444.439,E2 -22444.439} C_VEL
LIN {X 0,Y 201.204,Z 456.079,A -85,B 0,C 180,E1 -22445.651,E2 -22445.651} C_VEL
LIN {X 0,Y 203.082,Z 443.212,A -85,B 0,C 180,E1 -22446.523,E2 -22446.523} C_VEL
LIN {X 0,Y 204.162,Z 428.91,A -85,B 0,C 180,E1 -22447.117,E2 -22447.117} C_VEL
LIN {X 0,Y 205.885,Z 392.515,A -85,B 0,C 180,E1 -22448.317,E2 -22448.317} C_VEL
LIN {X 0,Y 203.751,Z 368.252,A -85,B 0,C 180,E1 -22449.866,E2 -22449.866} C_VEL
LIN {X 0,Y 200.239,Z 357.512,A -85,B 0,C 180,E1 -22451.2,E2 -22451.2} C_VEL
LIN {X 0,Y 194.376,Z 347.411,A -85,B 0,C 180,E1 -22453.215,E2 -22453.215} C_VEL
LIN {X 0,Y 187.252,Z 336.623,A -85,B 0,C 180,E1 -22455.859,E2 -22455.859} C_VEL
LIN {X 0,Y 184.313,Z 332.453,A -85,B 0,C 180,E1 -22457.032,E2 -22457.032} C_VEL
LIN {X 0,Y 182.069,Z 329.26,A -85,B 0,C 180,E1 -22457.973,E2 -22457.973} C_VEL
LIN {X 0,Y 181.352,Z 328.152,A -85,B 0,C 180,E1 -22458.287,E2 -22458.287} C_VEL
LIN {X 0,Y 179.376,Z 326.055,A -85,B 0,C 180,E1 -22459.119,E2 -22459.119} C_VEL
LIN {X 0,Y 178.499,Z 323.822,A -85,B 0,C 180,E1 -22459.577,E2 -22459.577} C_VEL
LIN {X 0,Y 178.426,Z 323.248,A -85,B 0,C 180,E1 -22459.696,E2 -22459.696} C_VEL
LIN {X 0,Y 178.476,Z 323.242,A -85,B 0,C 180,E1 -22465.781,E2 -22465.781} C_VEL
LIN {X 0,Y 178.474,Z 323.243,A -85,B 0,C 180,E1 -22470.029,E2 -22470.029} C_VEL
LIN {X 0,Y 178.498,Z 323.239,A -85,B 0,C 180,E1 -22474.895,E2 -22474.895} C_VEL
LIN {X 0,Y 178.6,Z 323.187,A -85,B 0,C 180,E1 -22481.651,E2 -22481.651} C_VEL
LIN {X 0,Y 178.637,Z 323.22,A -85,B 0,C 180,E1 -22486.346,E2 -22486.346} C_VEL
LIN {X 0,Y 178.896,Z 323.176,A -85,B 0,C 180,E1 -22490.959,E2 -22490.959} C_VEL
LIN {X 0,Y 179.115,Z 323.152,A -85,B 0,C 180,E1 -22497.751,E2 -22497.751} C_VEL
LIN {X 0,Y 179.336,Z 323.144,A -85,B 0,C 180,E1 -22500,E2 -22500} C_VEL
LIN {X 0,Y 178.821,Z 323.198,A -85,B 0,C 180,E1 -22504.508,E2 -22504.508} C_VEL
LIN {X 0,Y 178.896,Z 323.187,A -85,B 0,C 180,E1 -22509.041,E2 -22509.041} C_VEL
LIN {X 0,Y 178.637,Z 323.231,A -85,B 0,C 180,E1 -22513.654,E2 -22513.654} C_VEL
LIN {X 0,Y 178.583,Z 323.227,A -85,B 0,C 180,E1 -22519.187,E2 -22519.187} C_VEL
LIN {X 0,Y 178.509,Z 323.225,A -85,B 0,C 180,E1 -22525.112,E2 -22525.112} C_VEL
LIN {X 0,Y 178.454,Z 323.24,A -85,B 0,C 180,E1 -22530.796,E2 -22530.796} C_VEL
LIN {X 0,Y 178.477,Z 323.25,A -85,B 0,C 180,E1 -22534.22,E2 -22534.22} C_VEL
LIN {X 0,Y 178.39,Z 323.251,A -85,B 0,C 180,E1 -22539.076,E2 -22539.076} C_VEL
LIN {X 0,Y 178.421,Z 323.26,A -85,B 0,C 180,E1 -22540.789,E2 -22540.789} C_VEL
LIN {X 0,Y 179.277,Z 325.897,A -85,B 0,C 180,E1 -22541.277,E2 -22541.277} C_VEL
LIN {X 0,Y 181.324,Z 328.173,A -85,B 0,C 180,E1 -22542.146,E2 -22542.146} C_VEL
LIN {X 0,Y 182.231,Z 329.54,A -85,B 0,C 180,E1 -22542.541,E2 -22542.541} C_VEL
LIN {X 0,Y 184.49,Z 332.62,A -85,B 0,C 180,E1 -22543.478,E2 -22543.478} C_VEL
LIN {X 0,Y 191.198,Z 342.51,A -85,B 0,C 180,E1 -22546.085,E2 -22546.085} C_VEL
LIN {X 0,Y 198.42,Z 354.137,A -85,B 0,C 180,E1 -22548.63,E2 -22548.63} C_VEL
LIN {X 0,Y 206.26,Z 369.179,A -85,B 0,C 180,E1 -22551.202,E2 -22551.202} C_VEL
LIN {X 0,Y 207.444,Z 371.739,A -85,B 0,C 180,E1 -22551.578,E2 -22551.578} C_VEL
LIN {X 0,Y 204.713,Z 422.924,A -85,B 0,C 180,E1 -22553.277,E2 -22553.277} C_VEL
LIN {X 0,Y 203.411,Z 435.598,A -85,B 0,C 180,E1 -22554.033,E2 -22554.033} C_VEL
LIN {X 0,Y 201.448,Z 448.185,A -85,B 0,C 180,E1 -22555.163,E2 -22555.163} C_VEL
LIN {X 0,Y 199.173,Z 459.448,A -85,B 0,C 180,E1 -22556.544,E2 -22556.544} C_VEL
LIN {X 0,Y 196.512,Z 469.793,A -85,B 0,C 180,E1 -22558.165,E2 -22558.165} C_VEL
LIN {X 0,Y 193.353,Z 480.694,A -85,B 0,C 180,E1 -22560.407,E2 -22560.407} C_VEL
LIN {X 0,Y 190.562,Z 489.588,A -85,B 0,C 180,E1 -22562.746,E2 -22562.746} C_VEL
LIN {X 0,Y 187.244,Z 498.399,A -85,B 0,C 180,E1 -22565.617,E2 -22565.617} C_VEL
LIN {X 0,Y 184.224,Z 505.848,A -85,B 0,C 180,E1 -22568.754,E2 -22568.754} C_VEL
LIN {X 0,Y 181.72,Z 511.824,A -85,B 0,C 180,E1 -22571.979,E2 -22571.979} C_VEL
LIN {X 0,Y 179.724,Z 516.541,A -85,B 0,C 180,E1 -22575.278,E2 -22575.278} C_VEL
LIN {X 0,Y 178.264,Z 520.139,A -85,B 0,C 180,E1 -22578.634,E2 -22578.634} C_VEL
LIN {X 0,Y 177.533,Z 521.991,A -85,B 0,C 180,E1 -22580.891,E2 -22580.891} C_VEL
LIN {X 0,Y 176.961,Z 523.402,A -85,B 0,C 180,E1 -22583.16,E2 -22583.16} C_VEL
LIN {X 0,Y 176.424,Z 524.996,A -85,B 0,C 180,E1 -22587.719,E2 -22587.719} C_VEL
LIN {X 0,Y 176.362,Z 525.226,A -85,B 0,C 180,E1 -22590.002,E2 -22590.002} C_VEL
LIN {X 0,Y 176.424,Z 525.028,A -85,B 0,C 180,E1 -22592.285,E2 -22592.285} C_VEL
LIN {X 0,Y 176.962,Z 523.477,A -85,B 0,C 180,E1 -22596.845,E2 -22596.845} C_VEL
LIN {X 0,Y 177.53,Z 522.108,A -85,B 0,C 180,E1 -22599.113,E2 -22599.113} C_VEL
LIN {X 0,Y 178.615,Z 519.239,A -85,B 0,C 180,E1 -22602.5,E2 -22602.5} C_VEL
LIN {X 0,Y 180.286,Z 515.327,A -85,B 0,C 180,E1 -22605.838,E2 -22605.838} C_VEL
LIN {X 0,Y 182.46,Z 510.257,A -85,B 0,C 180,E1 -22609.113,E2 -22609.113} C_VEL
LIN {X 0,Y 185.043,Z 503.865,A -85,B 0,C 180,E1 -22612.324,E2 -22612.324} C_VEL
LIN {X 0,Y 188.328,Z 495.893,A -85,B 0,C 180,E1 -22615.416,E2 -22615.416} C_VEL
LIN {X 0,Y 191.177,Z 487.997,A -85,B 0,C 180,E1 -22617.864,E2 -22617.864} C_VEL
LIN {X 0,Y 194.031,Z 478.829,A -85,B 0,C 180,E1 -22620.172,E2 -22620.172} C_VEL
LIN {X 0,Y 197.185,Z 467.764,A -85,B 0,C 180,E1 -22622.321,E2 -22622.321} C_VEL
LIN {X 0,Y 199.884,Z 456.942,A -85,B 0,C 180,E1 -22623.932,E2 -22623.932} C_VEL
LIN {X 0,Y 202.126,Z 444.944,A -85,B 0,C 180,E1 -22625.316,E2 -22625.316} C_VEL
LIN {X 0,Y 204.033,Z 431.753,A -85,B 0,C 180,E1 -22626.363,E2 -22626.363} C_VEL
LIN {X 0,Y 205.208,Z 418.935,A -85,B 0,C 180,E1 -22627.015,E2 -22627.015} C_VEL
LIN {X 0,Y 207.567,Z 371.84,A -85,B 0,C 180,E1 -22628.559,E2 -22628.559} C_VEL
LIN {X 0,Y 199.825,Z 356.566,A -85,B 0,C 180,E1 -22631.076,E2 -22631.076} C_VEL
LIN {X 0,Y 192.578,Z 344.466,A -85,B 0,C 180,E1 -22633.607,E2 -22633.607} C_VEL
LIN {X 0,Y 186.876,Z 336.025,A -85,B 0,C 180,E1 -22635.763,E2 -22635.763} C_VEL
LIN {X 0,Y 184.379,Z 332.444,A -85,B 0,C 180,E1 -22636.771,E2 -22636.771} C_VEL
LIN {X 0,Y 182.142,Z 329.242,A -85,B 0,C 180,E1 -22637.714,E2 -22637.714} C_VEL
LIN {X 0,Y 181.36,Z 328.159,A -85,B 0,C 180,E1 -22638.051,E2 -22638.051} C_VEL
LIN {X 0,Y 179.345,Z 325.974,A -85,B 0,C 180,E1 -22638.908,E2 -22638.908} C_VEL
LIN {X 0,Y 178.43,Z 323.251,A -85,B 0,C 180,E1 -22639.465,E2 -22639.465} C_VEL
LIN {X 0,Y 178.428,Z 323.244,A -85,B 0,C 180,E1 -22643.784,E2 -22643.784} C_VEL
LIN {X 0,Y 178.492,Z 323.252,A -85,B 0,C 180,E1 -22646.548,E2 -22646.548} C_VEL
LIN {X 0,Y 178.665,Z 323.23,A -85,B 0,C 180,E1 -22652.446,E2 -22652.446} C_VEL
LIN {X 0,Y 185.688,Z 351.478,A -85,B 0,C 180,E1 -22654.681,E2 -22654.681} C_VEL
LIN {X 0,Y 182.192,Z 424.653,A -85,B 0,C 180,E1 -22659.98,E2 -22659.98} C_VEL
LIN {X 0,Y 181.208,Z 438.953,A -85,B 0,C 180,E1 -22661.485,E2 -22661.485} C_VEL
LIN {X 0,Y 180.363,Z 451.826,A -85,B 0,C 180,E1 -22663.299,E2 -22663.299} C_VEL
LIN {X 0,Y 179.378,Z 464.301,A -85,B 0,C 180,E1 -22665.536,E2 -22665.536} C_VEL
LIN {X 0,Y 178.432,Z 476.762,A -85,B 0,C 180,E1 -22668.354,E2 -22668.354} C_VEL
LIN {X 0,Y 177.761,Z 485.971,A -85,B 0,C 180,E1 -22670.901,E2 -22670.901} C_VEL
LIN {X 0,Y 177.266,Z 494.437,A -85,B 0,C 180,E1 -22673.706,E2 -22673.706} C_VEL
LIN {X 0,Y 176.951,Z 502.98,A -85,B 0,C 180,E1 -22677.154,E2 -22677.154} C_VEL
LIN {X 0,Y 176.749,Z 510.849,A -85,B 0,C 180,E1 -22681.139,E2 -22681.139} C_VEL
LIN {X 0,Y 177.025,Z 516.225,A -85,B 0,C 180,E1 -22684.554,E2 -22684.554} C_VEL
LIN {X 0,Y 177.835,Z 521.525,A -85,B 0,C 180,E1 -22688.876,E2 -22688.876} C_VEL
LIN {X 0,Y 180.083,Z 525.696,A -85,B 0,C 180,E1 -22693.542,E2 -22693.542} C_VEL
LIN {X 0,Y 183.412,Z 528.215,A -85,B 0,C 180,E1 -22697.851,E2 -22697.851} C_VEL
LIN {X 0,Y 185.442,Z 528.94,A -85,B 0,C 180,E1 -22699.943,E2 -22699.943} C_VEL
LIN {X 0,Y 190.587,Z 529.328,A -85,B 0,C 180,E1 -22703.931,E2 -22703.931} C_VEL
LIN {X 0,Y 196.793,Z 528.356,A -85,B 0,C 180,E1 -22707.663,E2 -22707.663} C_VEL
LIN {X 0,Y 204.047,Z 525.998,A -85,B 0,C 180,E1 -22711.108,E2 -22711.108} C_VEL
LIN {X 0,Y 212.248,Z 522.114,A -85,B 0,C 180,E1 -22714.257,E2 -22714.257} C_VEL
LIN {X 0,Y 219.568,Z 517.779,A -85,B 0,C 180,E1 -22716.623,E2 -22716.623} C_VEL
LIN {X 0,Y 228.487,Z 511.455,A -85,B 0,C 180,E1 -22719.091,E2 -22719.091} C_VEL
LIN {X 0,Y 237.425,Z 503.936,A -85,B 0,C 180,E1 -22721.195,E2 -22721.195} C_VEL
LIN {X 0,Y 245.419,Z 496.106,A -85,B 0,C 180,E1 -22722.853,E2 -22722.853} C_VEL
LIN {X 0,Y 252.377,Z 488.349,A -85,B 0,C 180,E1 -22724.121,E2 -22724.121} C_VEL
LIN {X 0,Y 251.791,Z 489.101,A -85,B 0,C 180,E1 -22724.322,E2 -22724.322} C_VEL
LIN {X 0,Y 242.228,Z 500.074,A -85,B 0,C 180,E1 -22725.864,E2 -22725.864} C_VEL
LIN {X 0,Y 236.506,Z 505.928,A -85,B 0,C 180,E1 -22726.938,E2 -22726.938} C_VEL
LIN {X 0,Y 232.494,Z 509.619,A -85,B 0,C 180,E1 -22727.539,E2 -22727.539} C_VEL
LIN {X 0,Y 224.979,Z 515.524,A -85,B 0,C 180,E1 -22728.252,E2 -22728.252} C_VEL
LIN {X 0,Y 217.375,Z 520.712,A -85,B 0,C 180,E1 -22729.11,E2 -22729.11} C_VEL
LIN {X 0,Y 213.28,Z 523.352,A -85,B 0,C 180,E1 -22729.946,E2 -22729.946} C_VEL
LIN {X 0,Y 203.707,Z 529.152,A -85,B 0,C 180,E1 -22732.858,E2 -22732.858} C_VEL
LIN {X 0,Y 197.228,Z 532.464,A -85,B 0,C 180,E1 -22735.238,E2 -22735.238} C_VEL
LIN {X 0,Y 189.423,Z 535.701,A -85,B 0,C 180,E1 -22738.704,E2 -22738.704} C_VEL
LIN {X 0,Y 185.989,Z 536.828,A -85,B 0,C 180,E1 -22740.576,E2 -22740.576} C_VEL
LIN {X 0,Y 180.239,Z 538.151,A -85,B 0,C 180,E1 -22744.599,E2 -22744.599} C_VEL
LIN {X 0,Y 175.59,Z 538.223,A -85,B 0,C 180,E1 -22748.884,E2 -22748.884} C_VEL
LIN {X 0,Y 172.377,Z 537.032,A -85,B 0,C 180,E1 -22753.415,E2 -22753.415} C_VEL
LIN {X 0,Y 170.731,Z 535.076,A -85,B 0,C 180,E1 -22757.668,E2 -22757.668} C_VEL
LIN {X 0,Y 169.815,Z 537.37,A -85,B 0,C 180,E1 -22760.469,E2 -22760.469} C_VEL
LIN {X 0,Y 169.353,Z 538.801,A -85,B 0,C 180,E1 -22762.846,E2 -22762.846} C_VEL
LIN {X 0,Y 169.129,Z 540.007,A -85,B 0,C 180,E1 -22765.787,E2 -22765.787} C_VEL
LIN {X 0,Y 169.329,Z 540.668,A -85,B 0,C 180,E1 -22769.998,E2 -22769.998} C_VEL
LIN {X 0,Y 169.045,Z 540.117,A -85,B 0,C 180,E1 -22773.806,E2 -22773.806} C_VEL
LIN {X 0,Y 169.086,Z 538.757,A -85,B 0,C 180,E1 -22777.161,E2 -22777.161} C_VEL
LIN {X 0,Y 169.345,Z 537.298,A -85,B 0,C 180,E1 -22779.553,E2 -22779.553} C_VEL
LIN {X 0,Y 170.151,Z 534.284,A -85,B 0,C 180,E1 -22783.128,E2 -22783.128} C_VEL
LIN {X 0,Y 171.629,Z 530.215,A -85,B 0,C 180,E1 -22786.654,E2 -22786.654} C_VEL
LIN {X 0,Y 174.141,Z 523.954,A -85,B 0,C 180,E1 -22790.677,E2 -22790.677} C_VEL
LIN {X 0,Y 176.727,Z 517.549,A -85,B 0,C 180,E1 -22793.843,E2 -22793.843} C_VEL
LIN {X 0,Y 179.576,Z 510.174,A -85,B 0,C 180,E1 -22796.746,E2 -22796.746} C_VEL
LIN {X 0,Y 182.785,Z 501.783,A -85,B 0,C 180,E1 -22799.353,E2 -22799.353} C_VEL
LIN {X 0,Y 186.427,Z 491.404,A -85,B 0,C 180,E1 -22801.853,E2 -22801.853} C_VEL
LIN {X 0,Y 189.995,Z 479.725,A -85,B 0,C 180,E1 -22804.017,E2 -22804.017} C_VEL
LIN {X 0,Y 192.997,Z 467.963,A -85,B 0,C 180,E1 -22805.634,E2 -22805.634} C_VEL
LIN {X 0,Y 195.488,Z 455.784,A -85,B 0,C 180,E1 -22806.862,E2 -22806.862} C_VEL
LIN {X 0,Y 197.347,Z 443.724,A -85,B 0,C 180,E1 -22807.703,E2 -22807.703} C_VEL
LIN {X 0,Y 198.493,Z 429.789,A -85,B 0,C 180,E1 -22808.315,E2 -22808.315} C_VEL
LIN {X 0,Y 200.333,Z 393.37,A -85,B 0,C 180,E1 -22809.534,E2 -22809.534} C_VEL
LIN {X 0,Y 198.326,Z 370.439,A -85,B 0,C 180,E1 -22811.074,E2 -22811.074} C_VEL
LIN {X 0,Y 195.522,Z 361.516,A -85,B 0,C 180,E1 -22812.218,E2 -22812.218} C_VEL
LIN {X 0,Y 189.646,Z 351.342,A -85,B 0,C 180,E1 -22814.36,E2 -22814.36} C_VEL
LIN {X 0,Y 183.202,Z 341.498,A -85,B 0,C 180,E1 -22816.896,E2 -22816.896} C_VEL
LIN {X 0,Y 180.427,Z 337.564,A -85,B 0,C 180,E1 -22818.066,E2 -22818.066} C_VEL
LIN {X 0,Y 177.652,Z 333.626,A -85,B 0,C 180,E1 -22819.302,E2 -22819.302} C_VEL
LIN {X 0,Y 175.405,Z 330.538,A -85,B 0,C 180,E1 -22820.348,E2 -22820.348} C_VEL
LIN {X 0,Y 174.537,Z 329.22,A -85,B 0,C 180,E1 -22820.774,E2 -22820.774} C_VEL
LIN {X 0,Y 172.446,Z 327.133,A -85,B 0,C 180,E1 -22821.763,E2 -22821.763} C_VEL
LIN {X 0,Y 171.458,Z 324.77,A -85,B 0,C 180,E1 -22822.338,E2 -22822.338} C_VEL
LIN {X 0,Y 171.36,Z 324.135,A -85,B 0,C 180,E1 -22822.498,E2 -22822.498} C_VEL
LIN {X 0,Y 171.402,Z 324.132,A -85,B 0,C 180,E1 -22827.789,E2 -22827.789} C_VEL
LIN {X 0,Y 171.401,Z 324.126,A -85,B 0,C 180,E1 -22830.525,E2 -22830.525} C_VEL
LIN {X 0,Y 171.42,Z 324.125,A -85,B 0,C 180,E1 -22835.796,E2 -22835.796} C_VEL
LIN {X 0,Y 171.499,Z 324.076,A -85,B 0,C 180,E1 -22840.862,E2 -22840.862} C_VEL
LIN {X 0,Y 171.551,Z 324.093,A -85,B 0,C 180,E1 -22845.771,E2 -22845.771} C_VEL
LIN {X 0,Y 171.835,Z 324.06,A -85,B 0,C 180,E1 -22850.584,E2 -22850.584} C_VEL
LIN {X 0,Y 171.773,Z 324.028,A -85,B 0,C 180,E1 -22855.306,E2 -22855.306} C_VEL
LIN {X 0,Y 172.301,Z 324.02,A -85,B 0,C 180,E1 -22860,E2 -22860} C_VEL
LIN {X 0,Y 171.837,Z 324.078,A -85,B 0,C 180,E1 -22866.919,E2 -22866.919} C_VEL
LIN {X 0,Y 171.76,Z 324.079,A -85,B 0,C 180,E1 -22870.895,E2 -22870.895} C_VEL
LIN {X 0,Y 171.515,Z 324.092,A -85,B 0,C 180,E1 -22876.669,E2 -22876.669} C_VEL
LIN {X 0,Y 171.508,Z 324.111,A -85,B 0,C 180,E1 -22879.535,E2 -22879.535} C_VEL
LIN {X 0,Y 171.437,Z 324.106,A -85,B 0,C 180,E1 -22885.6,E2 -22885.6} C_VEL
LIN {X 0,Y 171.411,Z 324.118,A -85,B 0,C 180,E1 -22890.574,E2 -22890.574} C_VEL
LIN {X 0,Y 171.387,Z 324.137,A -85,B 0,C 180,E1 -22895.036,E2 -22895.036} C_VEL
LIN {X 0,Y 171.396,Z 324.191,A -85,B 0,C 180,E1 -22898.038,E2 -22898.038} C_VEL
LIN {X 0,Y 172.191,Z 326.664,A -85,B 0,C 180,E1 -22898.541,E2 -22898.541} C_VEL
LIN {X 0,Y 174.131,Z 328.923,A -85,B 0,C 180,E1 -22899.486,E2 -22899.486} C_VEL
LIN {X 0,Y 175.033,Z 329.792,A -85,B 0,C 180,E1 -22899.901,E2 -22899.901} C_VEL
LIN {X 0,Y 177.104,Z 333.088,A -85,B 0,C 180,E1 -22900.904,E2 -22900.904} C_VEL
LIN {X 0,Y 178.599,Z 334.835,A -85,B 0,C 180,E1 -22901.563,E2 -22901.563} C_VEL
LIN {X 0,Y 184.573,Z 343.539,A -85,B 0,C 180,E1 -22904.11,E2 -22904.11} C_VEL
LIN {X 0,Y 190.938,Z 353.44,A -85,B 0,C 180,E1 -22906.57,E2 -22906.57} C_VEL
LIN {X 0,Y 197.373,Z 365.015,A -85,B 0,C 180,E1 -22908.88,E2 -22908.88} C_VEL
LIN {X 0,Y 201.761,Z 373.932,A -85,B 0,C 180,E1 -22910.375,E2 -22910.375} C_VEL
LIN {X 0,Y 199.081,Z 423.066,A -85,B 0,C 180,E1 -22912.051,E2 -22912.051} C_VEL
LIN {X 0,Y 197.723,Z 435.888,A -85,B 0,C 180,E1 -22912.827,E2 -22912.827} C_VEL
LIN {X 0,Y 195.66,Z 448.485,A -85,B 0,C 180,E1 -22913.975,E2 -22913.975} C_VEL
LIN {X 0,Y 193.302,Z 459.753,A -85,B 0,C 180,E1 -22915.386,E2 -22915.386} C_VEL
LIN {X 0,Y 190.542,Z 470.101,A -85,B 0,C 180,E1 -22917.044,E2 -22917.044} C_VEL
LIN {X 0,Y 187.317,Z 480.694,A -85,B 0,C 180,E1 -22919.259,E2 -22919.259} C_VEL
LIN {X 0,Y 184.219,Z 490.111,A -85,B 0,C 180,E1 -22921.8,E2 -22921.8} C_VEL
LIN {X 0,Y 180.819,Z 498.714,A -85,B 0,C 180,E1 -22924.691,E2 -22924.691} C_VEL
LIN {X 0,Y 177.604,Z 506.166,A -85,B 0,C 180,E1 -22927.921,E2 -22927.921} C_VEL
LIN {X 0,Y 174.984,Z 512.14,A -85,B 0,C 180,E1 -22931.26,E2 -22931.26} C_VEL
LIN {X 0,Y 172.885,Z 516.857,A -85,B 0,C 180,E1 -22934.681,E2 -22934.681} C_VEL
LIN {X 0,Y 171.3,Z 520.457,A -85,B 0,C 180,E1 -22938.165,E2 -22938.165} C_VEL
LIN {X 0,Y 170.532,Z 522.308,A -85,B 0,C 180,E1 -22940.514,E2 -22940.514} C_VEL
LIN {X 0,Y 169.819,Z 523.935,A -85,B 0,C 180,E1 -22943.34,E2 -22943.34} C_VEL
LIN {X 0,Y 169.352,Z 525.313,A -85,B 0,C 180,E1 -22947.624,E2 -22947.624} C_VEL
LIN {X 0,Y 169.284,Z 525.542,A -85,B 0,C 180,E1 -22950.002,E2 -22950.002} C_VEL
LIN {X 0,Y 169.352,Z 525.344,A -85,B 0,C 180,E1 -22952.381,E2 -22952.381} C_VEL
LIN {X 0,Y 169.927,Z 523.793,A -85,B 0,C 180,E1 -22957.13,E2 -22957.13} C_VEL
LIN {X 0,Y 170.526,Z 522.424,A -85,B 0,C 180,E1 -22959.491,E2 -22959.491} C_VEL
LIN {X 0,Y 171.688,Z 519.555,A -85,B 0,C 180,E1 -22963.013,E2 -22963.013} C_VEL
LIN {X 0,Y 173.467,Z 515.642,A -85,B 0,C 180,E1 -22966.478,E2 -22966.478} C_VEL
LIN {X 0,Y 175.776,Z 510.57,A -85,B 0,C 180,E1 -22969.87,E2 -22969.87} C_VEL
LIN {X 0,Y 178.504,Z 504.177,A -85,B 0,C 180,E1 -22973.188,E2 -22973.188} C_VEL
LIN {X 0,Y 181.955,Z 496.203,A -85,B 0,C 180,E1 -22976.374,E2 -22976.374} C_VEL
LIN {X 0,Y 184.769,Z 488.764,A -85,B 0,C 180,E1 -22978.755,E2 -22978.755} C_VEL
LIN {X 0,Y 187.938,Z 479.133,A -85,B 0,C 180,E1 -22981.258,E2 -22981.258} C_VEL
LIN {X 0,Y 191.245,Z 468.064,A -85,B 0,C 180,E1 -22983.454,E2 -22983.454} C_VEL
LIN {X 0,Y 194.047,Z 457.235,A -85,B 0,C 180,E1 -22985.099,E2 -22985.099} C_VEL
LIN {X 0,Y 196.399,Z 445.224,A -85,B 0,C 180,E1 -22986.509,E2 -22986.509} C_VEL
LIN {X 0,Y 198.381,Z 431.889,A -85,B 0,C 180,E1 -22987.586,E2 -22987.586} C_VEL
LIN {X 0,Y 199.587,Z 419.149,A -85,B 0,C 180,E1 -22988.241,E2 -22988.241} C_VEL
LIN {X 0,Y 201.948,Z 374.197,A -85,B 0,C 180,E1 -22989.743,E2 -22989.743} C_VEL
LIN {X 0,Y 195.082,Z 360.511,A -85,B 0,C 180,E1 -22992.117,E2 -22992.117} C_VEL
LIN {X 0,Y 187.804,Z 348.356,A -85,B 0,C 180,E1 -22994.813,E2 -22994.813} C_VEL
LIN {X 0,Y 182.776,Z 340.821,A -85,B 0,C 180,E1 -22996.836,E2 -22996.836} C_VEL
LIN {X 0,Y 180.551,Z 337.589,A -85,B 0,C 180,E1 -22997.786,E2 -22997.786} C_VEL
LIN {X 0,Y 177.947,Z 333.856,A -85,B 0,C 180,E1 -22998.95,E2 -22998.95} C_VEL
LIN {X 0,Y 175.589,Z 330.887,A -85,B 0,C 180,E1 -23000.033,E2 -23000.033} C_VEL
LIN {X 0,Y 174.648,Z 329.288,A -85,B 0,C 180,E1 -23000.507,E2 -23000.507} C_VEL
LIN {X 0,Y 172.574,Z 327.291,A -85,B 0,C 180,E1 -23001.487,E2 -23001.487} C_VEL
LIN {X 0,Y 171.45,Z 324.523,A -85,B 0,C 180,E1 -23002.15,E2 -23002.15} C_VEL
LIN {X 0,Y 171.403,Z 324.122,A -85,B 0,C 180,E1 -23002.231,E2 -23002.231} C_VEL
LIN {X 0,Y 171.422,Z 324.119,A -85,B 0,C 180,E1 -23007.793,E2 -23007.793} C_VEL
LIN {X 0,Y 171.593,Z 324.111,A -85,B 0,C 180,E1 -23012.303,E2 -23012.303} C_VEL
LIN {X 0,Y 176.082,Z 342.226,A -85,B 0,C 180,E1 -23013.789,E2 -23013.789} C_VEL
LIN {X 0,Y 178.534,Z 352.185,A -85,B 0,C 180,E1 -23014.581,E2 -23014.581} C_VEL
LIN {X 0,Y 175.054,Z 424.812,A -85,B 0,C 180,E1 -23020.123,E2 -23020.123} C_VEL
LIN {X 0,Y 174.082,Z 439.614,A -85,B 0,C 180,E1 -23021.767,E2 -23021.767} C_VEL
LIN {X 0,Y 173.199,Z 453.203,A -85,B 0,C 180,E1 -23023.801,E2 -23023.801} C_VEL
LIN {X 0,Y 172.203,Z 465.365,A -85,B 0,C 180,E1 -23026.127,E2 -23026.127} C_VEL
LIN {X 0,Y 171.288,Z 477.609,A -85,B 0,C 180,E1 -23029.061,E2 -23029.061} C_VEL
LIN {X 0,Y 170.656,Z 487.348,A -85,B 0,C 180,E1 -23031.923,E2 -23031.923} C_VEL
LIN {X 0,Y 170.129,Z 496.592,A -85,B 0,C 180,E1 -23035.261,E2 -23035.261} C_VEL
LIN {X 0,Y 169.917,Z 504.683,A -85,B 0,C 180,E1 -23038.815,E2 -23038.815} C_VEL
LIN {X 0,Y 169.844,Z 511.226,A -85,B 0,C 180,E1 -23042.371,E2 -23042.371} C_VEL
LIN {X 0,Y 170.222,Z 516.554,A -85,B 0,C 180,E1 -23045.924,E2 -23045.924} C_VEL
LIN {X 0,Y 170.962,Z 520.83,A -85,B 0,C 180,E1 -23049.464,E2 -23049.464} C_VEL
LIN {X 0,Y 173.217,Z 525.216,A -85,B 0,C 180,E1 -23054.09,E2 -23054.09} C_VEL
LIN {X 0,Y 176.673,Z 528.105,A -85,B 0,C 180,E1 -23058.556,E2 -23058.556} C_VEL
LIN {X 0,Y 181.334,Z 529.631,A -85,B 0,C 180,E1 -23062.803,E2 -23062.803} C_VEL
LIN {X 0,Y 187.235,Z 529.817,A -85,B 0,C 180,E1 -23066.771,E2 -23066.771} C_VEL
LIN {X 0,Y 194.285,Z 528.644,A -85,B 0,C 180,E1 -23070.426,E2 -23070.426} C_VEL
LIN {X 0,Y 202.259,Z 526.063,A -85,B 0,C 180,E1 -23073.777,E2 -23073.777} C_VEL
LIN {X 0,Y 211.16,Z 522.021,A -85,B 0,C 180,E1 -23076.805,E2 -23076.805} C_VEL
LIN {X 0,Y 220.855,Z 516.395,A -85,B 0,C 180,E1 -23079.527,E2 -23079.527} C_VEL
LIN {X 0,Y 229.903,Z 510.01,A -85,B 0,C 180,E1 -23081.674,E2 -23081.674} C_VEL
LIN {X 0,Y 239.414,Z 502.119,A -85,B 0,C 180,E1 -23083.618,E2 -23083.618} C_VEL
LIN {X 0,Y 240.708,Z 500.921,A -85,B 0,C 180,E1 -23083.867,E2 -23083.867} C_VEL
LIN {X 0,Y 239.374,Z 502.301,A -85,B 0,C 180,E1 -23084.408,E2 -23084.408} C_VEL
LIN {X 0,Y 228.896,Z 511.73,A -85,B 0,C 180,E1 -23086.301,E2 -23086.301} C_VEL
LIN {X 0,Y 220.775,Z 518.112,A -85,B 0,C 180,E1 -23088.046,E2 -23088.046} C_VEL
LIN {X 0,Y 213.28,Z 523.352,A -85,B 0,C 180,E1 -23089.946,E2 -23089.946} C_VEL
LIN {X 0,Y 209.115,Z 525.87,A -85,B 0,C 180,E1 -23090.87,E2 -23090.87} C_VEL
LIN {X 0,Y 197.949,Z 530.976,A -85,B 0,C 180,E1 -23092.705,E2 -23092.705} C_VEL
LIN {X 0,Y 191.901,Z 533.176,A -85,B 0,C 180,E1 -23094.028,E2 -23094.028} C_VEL
LIN {X 0,Y 189.366,Z 534.026,A -85,B 0,C 180,E1 -23094.88,E2 -23094.88} C_VEL
LIN {X 0,Y 183.421,Z 535.978,A -85,B 0,C 180,E1 -23097.557,E2 -23097.557} C_VEL
LIN {X 0,Y 179.85,Z 536.862,A -85,B 0,C 180,E1 -23099.467,E2 -23099.467} C_VEL
LIN {X 0,Y 173.864,Z 537.729,A -85,B 0,C 180,E1 -23103.597,E2 -23103.597} C_VEL
LIN {X 0,Y 169.025,Z 537.379,A -85,B 0,C 180,E1 -23108.022,E2 -23108.022} C_VEL
LIN {X 0,Y 165.674,Z 535.822,A -85,B 0,C 180,E1 -23112.723,E2 -23112.723} C_VEL
LIN {X 0,Y 164.261,Z 533.928,A -85,B 0,C 180,E1 -23116.229,E2 -23116.229} C_VEL
LIN {X 0,Y 162.801,Z 537.053,A -85,B 0,C 180,E1 -23120.054,E2 -23120.054} C_VEL
LIN {X 0,Y 162.301,Z 538.484,A -85,B 0,C 180,E1 -23122.533,E2 -23122.533} C_VEL
LIN {X 0,Y 162.042,Z 539.812,A -85,B 0,C 180,E1 -23125.986,E2 -23125.986} C_VEL
LIN {X 0,Y 162.243,Z 540.352,A -85,B 0,C 180,E1 -23129.998,E2 -23129.998} C_VEL
LIN {X 0,Y 161.965,Z 539.885,A -85,B 0,C 180,E1 -23133.605,E2 -23133.605} C_VEL
LIN {X 0,Y 162.004,Z 538.438,A -85,B 0,C 180,E1 -23137.475,E2 -23137.475} C_VEL
LIN {X 0,Y 162.323,Z 536.979,A -85,B 0,C 180,E1 -23139.97,E2 -23139.97} C_VEL
LIN {X 0,Y 163.208,Z 533.965,A -85,B 0,C 180,E1 -23143.697,E2 -23143.697} C_VEL
LIN {X 0,Y 164.796,Z 529.896,A -85,B 0,C 180,E1 -23147.366,E2 -23147.366} C_VEL
LIN {X 0,Y 167.508,Z 523.637,A -85,B 0,C 180,E1 -23151.535,E2 -23151.535} C_VEL
LIN {X 0,Y 170.355,Z 516.942,A -85,B 0,C 180,E1 -23154.947,E2 -23154.947} C_VEL
LIN {X 0,Y 173.236,Z 509.857,A -85,B 0,C 180,E1 -23157.807,E2 -23157.807} C_VEL
LIN {X 0,Y 176.598,Z 501.468,A -85,B 0,C 180,E1 -23160.488,E2 -23160.488} C_VEL
LIN {X 0,Y 180.418,Z 491.092,A -85,B 0,C 180,E1 -23163.046,E2 -23163.046} C_VEL
LIN {X 0,Y 184.154,Z 479.417,A -85,B 0,C 180,E1 -23165.253,E2 -23165.253} C_VEL
LIN {X 0,Y 187.266,Z 467.66,A -85,B 0,C 180,E1 -23166.901,E2 -23166.901} C_VEL
LIN {X 0,Y 189.865,Z 455.49,A -85,B 0,C 180,E1 -23168.145,E2 -23168.145} C_VEL
LIN {X 0,Y 191.892,Z 442.583,A -85,B 0,C 180,E1 -23169.045,E2 -23169.045} C_VEL
LIN {X 0,Y 192.987,Z 429.376,A -85,B 0,C 180,E1 -23169.627,E2 -23169.627} C_VEL
LIN {X 0,Y 194.865,Z 394.383,A -85,B 0,C 180,E1 -23170.815,E2 -23170.815} C_VEL
LIN {X 0,Y 193.121,Z 372.902,A -85,B 0,C 180,E1 -23172.303,E2 -23172.303} C_VEL
LIN {X 0,Y 190.716,Z 365.156,A -85,B 0,C 180,E1 -23173.348,E2 -23173.348} C_VEL
LIN {X 0,Y 183.7,Z 353.182,A -85,B 0,C 180,E1 -23176.087,E2 -23176.087} C_VEL
LIN {X 0,Y 177.133,Z 343.273,A -85,B 0,C 180,E1 -23178.913,E2 -23178.913} C_VEL
LIN {X 0,Y 173.955,Z 338.865,A -85,B 0,C 180,E1 -23180.396,E2 -23180.396} C_VEL
LIN {X 0,Y 171.287,Z 335.037,A -85,B 0,C 180,E1 -23181.73,E2 -23181.73} C_VEL
LIN {X 0,Y 168.87,Z 332.085,A -85,B 0,C 180,E1 -23182.975,E2 -23182.975} C_VEL
LIN {X 0,Y 167.857,Z 330.303,A -85,B 0,C 180,E1 -23183.557,E2 -23183.557} C_VEL
LIN {X 0,Y 165.579,Z 328.221,A -85,B 0,C 180,E1 -23184.782,E2 -23184.782} C_VEL
LIN {X 0,Y 164.454,Z 325.673,A -85,B 0,C 180,E1 -23185.527,E2 -23185.527} C_VEL
LIN {X 0,Y 164.327,Z 325.003,A -85,B 0,C 180,E1 -23185.704,E2 -23185.704} C_VEL
LIN {X 0,Y 164.363,Z 325,A -85,B 0,C 180,E1 -23189.129,E2 -23189.129} C_VEL
LIN {X 0,Y 164.379,Z 324.997,A -85,B 0,C 180,E1 -23194.688,E2 -23194.688} C_VEL
LIN {X 0,Y 164.409,Z 324.967,A -85,B 0,C 180,E1 -23200.117,E2 -23200.117} C_VEL
LIN {X 0,Y 164.478,Z 324.959,A -85,B 0,C 180,E1 -23205.145,E2 -23205.145} C_VEL
LIN {X 0,Y 164.756,Z 324.945,A -85,B 0,C 180,E1 -23210.176,E2 -23210.176} C_VEL
LIN {X 0,Y 164.811,Z 324.898,A -85,B 0,C 180,E1 -23212.65,E2 -23212.65} C_VEL
LIN {X 0,Y 165.265,Z 324.897,A -85,B 0,C 180,E1 -23220,E2 -23220} C_VEL
LIN {X 0,Y 164.811,Z 324.953,A -85,B 0,C 180,E1 -23227.35,E2 -23227.35} C_VEL
LIN {X 0,Y 164.694,Z 324.959,A -85,B 0,C 180,E1 -23231.059,E2 -23231.059} C_VEL
LIN {X 0,Y 164.444,Z 324.971,A -85,B 0,C 180,E1 -23237.408,E2 -23237.408} C_VEL
LIN {X 0,Y 164.442,Z 324.995,A -85,B 0,C 180,E1 -23239.993,E2 -23239.993} C_VEL
LIN {X 0,Y 164.364,Z 324.989,A -85,B 0,C 180,E1 -23246.118,E2 -23246.118} C_VEL
LIN {X 0,Y 164.347,Z 324.993,A -85,B 0,C 180,E1 -23251.216,E2 -23251.216} C_VEL
LIN {X 0,Y 164.34,Z 325.021,A -85,B 0,C 180,E1 -23254.807,E2 -23254.807} C_VEL
LIN {X 0,Y 165.24,Z 327.733,A -85,B 0,C 180,E1 -23255.458,E2 -23255.458} C_VEL
LIN {X 0,Y 167.273,Z 329.955,A -85,B 0,C 180,E1 -23256.591,E2 -23256.591} C_VEL
LIN {X 0,Y 168.237,Z 330.811,A -85,B 0,C 180,E1 -23257.094,E2 -23257.094} C_VEL
LIN {X 0,Y 170.319,Z 334.107,A -85,B 0,C 180,E1 -23258.24,E2 -23258.24} C_VEL
LIN {X 0,Y 171.916,Z 335.875,A -85,B 0,C 180,E1 -23259.031,E2 -23259.031} C_VEL
LIN {X 0,Y 174.512,Z 339.49,A -85,B 0,C 180,E1 -23260.307,E2 -23260.307} C_VEL
LIN {X 0,Y 180.411,Z 348.045,A -85,B 0,C 180,E1 -23262.979,E2 -23262.979} C_VEL
LIN {X 0,Y 186.98,Z 358.592,A -85,B 0,C 180,E1 -23265.674,E2 -23265.674} C_VEL
LIN {X 0,Y 192.942,Z 369.528,A -85,B 0,C 180,E1 -23267.935,E2 -23267.935} C_VEL
LIN {X 0,Y 196.259,Z 376.248,A -85,B 0,C 180,E1 -23269.131,E2 -23269.131} C_VEL
LIN {X 0,Y 193.55,Z 423.402,A -85,B 0,C 180,E1 -23270.767,E2 -23270.767} C_VEL
LIN {X 0,Y 192.131,Z 436.176,A -85,B 0,C 180,E1 -23271.552,E2 -23271.552} C_VEL
LIN {X 0,Y 189.973,Z 448.785,A -85,B 0,C 180,E1 -23272.717,E2 -23272.717} C_VEL
LIN {X 0,Y 187.517,Z 460.059,A -85,B 0,C 180,E1 -23274.157,E2 -23274.157} C_VEL
LIN {X 0,Y 184.647,Z 470.409,A -85,B 0,C 180,E1 -23275.849,E2 -23275.849} C_VEL
LIN {X 0,Y 181.251,Z 481.006,A -85,B 0,C 180,E1 -23278.112,E2 -23278.112} C_VEL
LIN {X 0,Y 177.936,Z 490.611,A -85,B 0,C 180,E1 -23280.779,E2 -23280.779} C_VEL
LIN {X 0,Y 174.444,Z 499.029,A -85,B 0,C 180,E1 -23283.697,E2 -23283.697} C_VEL
LIN {X 0,Y 171.046,Z 506.482,A -85,B 0,C 180,E1 -23287.027,E2 -23287.027} C_VEL
LIN {X 0,Y 168.285,Z 512.457,A -85,B 0,C 180,E1 -23290.485,E2 -23290.485} C_VEL
LIN {X 0,Y 166.041,Z 517.174,A -85,B 0,C 180,E1 -23294.033,E2 -23294.033} C_VEL
LIN {X 0,Y 164.348,Z 520.775,A -85,B 0,C 180,E1 -23297.657,E2 -23297.657} C_VEL
LIN {X 0,Y 163.529,Z 522.626,A -85,B 0,C 180,E1 -23300.104,E2 -23300.104} C_VEL
LIN {X 0,Y 162.684,Z 524.461,A -85,B 0,C 180,E1 -23303.522,E2 -23303.522} C_VEL
LIN {X 0,Y 162.262,Z 525.63,A -85,B 0,C 180,E1 -23307.52,E2 -23307.52} C_VEL
LIN {X 0,Y 162.209,Z 525.858,A -85,B 0,C 180,E1 -23310.002,E2 -23310.002} C_VEL
LIN {X 0,Y 162.262,Z 525.661,A -85,B 0,C 180,E1 -23312.485,E2 -23312.485} C_VEL
LIN {X 0,Y 162.898,Z 524.109,A -85,B 0,C 180,E1 -23317.439,E2 -23317.439} C_VEL
LIN {X 0,Y 163.522,Z 522.741,A -85,B 0,C 180,E1 -23319.902,E2 -23319.902} C_VEL
LIN {X 0,Y 164.786,Z 519.87,A -85,B 0,C 180,E1 -23323.569,E2 -23323.569} C_VEL
LIN {X 0,Y 166.664,Z 515.957,A -85,B 0,C 180,E1 -23327.171,E2 -23327.171} C_VEL
LIN {X 0,Y 169.126,Z 510.883,A -85,B 0,C 180,E1 -23330.687,E2 -23330.687} C_VEL
LIN {X 0,Y 172.016,Z 504.489,A -85,B 0,C 180,E1 -23334.117,E2 -23334.117} C_VEL
LIN {X 0,Y 175.638,Z 496.513,A -85,B 0,C 180,E1 -23337.4,E2 -23337.4} C_VEL
LIN {X 0,Y 178.411,Z 489.527,A -85,B 0,C 180,E1 -23339.711,E2 -23339.711} C_VEL
LIN {X 0,Y 181.911,Z 479.437,A -85,B 0,C 180,E1 -23342.418,E2 -23342.418} C_VEL
LIN {X 0,Y 185.387,Z 468.362,A -85,B 0,C 180,E1 -23344.658,E2 -23344.658} C_VEL
LIN {X 0,Y 188.288,Z 457.528,A -85,B 0,C 180,E1 -23346.34,E2 -23346.34} C_VEL
LIN {X 0,Y 190.763,Z 445.503,A -85,B 0,C 180,E1 -23347.772,E2 -23347.772} C_VEL
LIN {X 0,Y 192.764,Z 432.556,A -85,B 0,C 180,E1 -23348.843,E2 -23348.843} C_VEL
LIN {X 0,Y 194.049,Z 419.728,A -85,B 0,C 180,E1 -23349.52,E2 -23349.52} C_VEL
LIN {X 0,Y 196.421,Z 376.535,A -85,B 0,C 180,E1 -23350.994,E2 -23350.994} C_VEL
LIN {X 0,Y 189.692,Z 363.221,A -85,B 0,C 180,E1 -23353.477,E2 -23353.477} C_VEL
LIN {X 0,Y 182.691,Z 351.424,A -85,B 0,C 180,E1 -23356.267,E2 -23356.267} C_VEL
LIN {X 0,Y 176.794,Z 342.707,A -85,B 0,C 180,E1 -23358.843,E2 -23358.843} C_VEL
LIN {X 0,Y 174.151,Z 339.015,A -85,B 0,C 180,E1 -23360.088,E2 -23360.088} C_VEL
LIN {X 0,Y 171.165,Z 334.927,A -85,B 0,C 180,E1 -23361.576,E2 -23361.576} C_VEL
LIN {X 0,Y 168.853,Z 332.021,A -85,B 0,C 180,E1 -23362.784,E2 -23362.784} C_VEL
LIN {X 0,Y 167.842,Z 330.273,A -85,B 0,C 180,E1 -23363.367,E2 -23363.367} C_VEL
LIN {X 0,Y 165.653,Z 328.276,A -85,B 0,C 180,E1 -23364.552,E2 -23364.552} C_VEL
LIN {X 0,Y 164.482,Z 325.738,A -85,B 0,C 180,E1 -23365.324,E2 -23365.324} C_VEL
LIN {X 0,Y 164.349,Z 325.009,A -85,B 0,C 180,E1 -23365.501,E2 -23365.501} C_VEL
LIN {X 0,Y 164.57,Z 324.985,A -85,B 0,C 180,E1 -23372.094,E2 -23372.094} C_VEL
LIN {X 0,Y 167.655,Z 338.199,A -85,B 0,C 180,E1 -23373.284,E2 -23373.284} C_VEL
LIN {X 0,Y 171.375,Z 353.122,A -85,B 0,C 180,E1 -23374.523,E2 -23374.523} C_VEL
LIN {X 0,Y 167.924,Z 425.483,A -85,B 0,C 180,E1 -23380.359,E2 -23380.359} C_VEL
LIN {X 0,Y 166.968,Z 440.049,A -85,B 0,C 180,E1 -23382.073,E2 -23382.073} C_VEL
LIN {X 0,Y 166.043,Z 454.361,A -85,B 0,C 180,E1 -23384.346,E2 -23384.346} C_VEL
LIN {X 0,Y 164.969,Z 467.596,A -85,B 0,C 180,E1 -23387.076,E2 -23387.076} C_VEL
LIN {X 0,Y 164.144,Z 478.919,A -85,B 0,C 180,E1 -23389.999,E2 -23389.999} C_VEL
LIN {X 0,Y 163.556,Z 489.047,A -85,B 0,C 180,E1 -23393.214,E2 -23393.214} C_VEL
LIN {X 0,Y 163.12,Z 498.523,A -85,B 0,C 180,E1 -23396.913,E2 -23396.913} C_VEL
LIN {X 0,Y 162.953,Z 505.032,A -85,B 0,C 180,E1 -23400,E2 -23400} C_VEL
LIN {X 0,Y 163.024,Z 511.516,A -85,B 0,C 180,E1 -23403.708,E2 -23403.708} C_VEL
LIN {X 0,Y 163.463,Z 516.794,A -85,B 0,C 180,E1 -23407.411,E2 -23407.411} C_VEL
LIN {X 0,Y 165.044,Z 522.352,A -85,B 0,C 180,E1 -23412.293,E2 -23412.293} C_VEL
LIN {X 0,Y 168.066,Z 526.367,A -85,B 0,C 180,E1 -23417.021,E2 -23417.021} C_VEL
LIN {X 0,Y 172.181,Z 529.002,A -85,B 0,C 180,E1 -23421.553,E2 -23421.553} C_VEL
LIN {X 0,Y 177.769,Z 530.322,A -85,B 0,C 180,E1 -23425.778,E2 -23425.778} C_VEL
LIN {X 0,Y 184.476,Z 530.3,A -85,B 0,C 180,E1 -23429.687,E2 -23429.687} C_VEL
LIN {X 0,Y 192.288,Z 528.918,A -85,B 0,C 180,E1 -23433.246,E2 -23433.246} C_VEL
LIN {X 0,Y 201.046,Z 526.176,A -85,B 0,C 180,E1 -23436.461,E2 -23436.461} C_VEL
LIN {X 0,Y 208.17,Z 523.172,A -85,B 0,C 180,E1 -23438.651,E2 -23438.651} C_VEL
LIN {X 0,Y 218.322,Z 517.82,A -85,B 0,C 180,E1 -23441.294,E2 -23441.294} C_VEL
LIN {X 0,Y 228.175,Z 511.43,A -85,B 0,C 180,E1 -23443.441,E2 -23443.441} C_VEL
LIN {X 0,Y 229.22,Z 510.666,A -85,B 0,C 180,E1 -23443.643,E2 -23443.643} C_VEL
LIN {X 0,Y 229.655,Z 510.412,A -85,B 0,C 180,E1 -23444.067,E2 -23444.067} C_VEL
LIN {X 0,Y 221.218,Z 516.776,A -85,B 0,C 180,E1 -23445.657,E2 -23445.657} C_VEL
LIN {X 0,Y 213.034,Z 522.225,A -85,B 0,C 180,E1 -23447.443,E2 -23447.443} C_VEL
LIN {X 0,Y 202.897,Z 528.026,A -85,B 0,C 180,E1 -23450.146,E2 -23450.146} C_VEL
LIN {X 0,Y 195.898,Z 531.433,A -85,B 0,C 180,E1 -23452.416,E2 -23452.416} C_VEL
LIN {X 0,Y 189.366,Z 534.026,A -85,B 0,C 180,E1 -23454.88,E2 -23454.88} C_VEL
LIN {X 0,Y 186.544,Z 534.899,A -85,B 0,C 180,E1 -23455.715,E2 -23455.715} C_VEL
LIN {X 0,Y 175.664,Z 536.605,A -85,B 0,C 180,E1 -23457.809,E2 -23457.809} C_VEL
LIN {X 0,Y 173.011,Z 536.853,A -85,B 0,C 180,E1 -23458.771,E2 -23458.771} C_VEL
LIN {X 0,Y 172.682,Z 536.863,A -85,B 0,C 180,E1 -23458.96,E2 -23458.96} C_VEL
LIN {X 0,Y 167.548,Z 537.161,A -85,B 0,C 180,E1 -23462.519,E2 -23462.519} C_VEL
LIN {X 0,Y 162.508,Z 536.392,A -85,B 0,C 180,E1 -23467.091,E2 -23467.091} C_VEL
LIN {X 0,Y 159.014,Z 534.448,A -85,B 0,C 180,E1 -23471.975,E2 -23471.975} C_VEL
LIN {X 0,Y 157.774,Z 532.836,A -85,B 0,C 180,E1 -23474.826,E2 -23474.826} C_VEL
LIN {X 0,Y 155.81,Z 536.737,A -85,B 0,C 180,E1 -23479.603,E2 -23479.603} C_VEL
LIN {X 0,Y 155.246,Z 538.167,A -85,B 0,C 180,E1 -23482.192,E2 -23482.192} C_VEL
LIN {X 0,Y 154.947,Z 539.591,A -85,B 0,C 180,E1 -23486.258,E2 -23486.258} C_VEL
LIN {X 0,Y 155.157,Z 540.035,A -85,B 0,C 180,E1 -23489.997,E2 -23489.997} C_VEL
LIN {X 0,Y 154.897,Z 539.63,A -85,B 0,C 180,E1 -23493.448,E2 -23493.448} C_VEL
LIN {X 0,Y 154.946,Z 538.119,A -85,B 0,C 180,E1 -23497.818,E2 -23497.818} C_VEL
LIN {X 0,Y 155.287,Z 536.659,A -85,B 0,C 180,E1 -23500.427,E2 -23500.427} C_VEL
LIN {X 0,Y 156.262,Z 533.645,A -85,B 0,C 180,E1 -23504.319,E2 -23504.319} C_VEL
LIN {X 0,Y 157.996,Z 529.577,A -85,B 0,C 180,E1 -23508.139,E2 -23508.139} C_VEL
LIN {X 0,Y 160.921,Z 523.32,A -85,B 0,C 180,E1 -23512.464,E2 -23512.464} C_VEL
LIN {X 0,Y 163.952,Z 516.499,A -85,B 0,C 180,E1 -23516.061,E2 -23516.061} C_VEL
LIN {X 0,Y 166.958,Z 509.541,A -85,B 0,C 180,E1 -23518.95,E2 -23518.95} C_VEL
LIN {X 0,Y 170.496,Z 501.153,A -85,B 0,C 180,E1 -23521.703,E2 -23521.703} C_VEL
LIN {X 0,Y 174.499,Z 490.78,A -85,B 0,C 180,E1 -23524.32,E2 -23524.32} C_VEL
LIN {X 0,Y 178.399,Z 479.109,A -85,B 0,C 180,E1 -23526.57,E2 -23526.57} C_VEL
LIN {X 0,Y 181.644,Z 467.358,A -85,B 0,C 180,E1 -23528.244,E2 -23528.244} C_VEL
LIN {X 0,Y 184.33,Z 455.196,A -85,B 0,C 180,E1 -23529.509,E2 -23529.509} C_VEL
LIN {X 0,Y 186.41,Z 442.576,A -85,B 0,C 180,E1 -23530.403,E2 -23530.403} C_VEL
LIN {X 0,Y 187.598,Z 428.705,A -85,B 0,C 180,E1 -23531.026,E2 -23531.026} C_VEL
LIN {X 0,Y 189.494,Z 395.047,A -85,B 0,C 180,E1 -23532.188,E2 -23532.188} C_VEL
LIN {X 0,Y 187.919,Z 374.976,A -85,B 0,C 180,E1 -23533.645,E2 -23533.645} C_VEL
LIN {X 0,Y 186.027,Z 369,A -85,B 0,C 180,E1 -23534.513,E2 -23534.513} C_VEL
LIN {X 0,Y 179.371,Z 357.476,A -85,B 0,C 180,E1 -23537.283,E2 -23537.283} C_VEL
LIN {X 0,Y 173.494,Z 348.49,A -85,B 0,C 180,E1 -23539.972,E2 -23539.972} C_VEL
LIN {X 0,Y 170.292,Z 343.947,A -85,B 0,C 180,E1 -23541.561,E2 -23541.561} C_VEL
LIN {X 0,Y 167.698,Z 340.326,A -85,B 0,C 180,E1 -23542.932,E2 -23542.932} C_VEL
LIN {X 0,Y 165.281,Z 336.854,A -85,B 0,C 180,E1 -23544.297,E2 -23544.297} C_VEL
LIN {X 0,Y 162.32,Z 333.454,A -85,B 0,C 180,E1 -23546.027,E2 -23546.027} C_VEL
LIN {X 0,Y 161.187,Z 331.389,A -85,B 0,C 180,E1 -23546.788,E2 -23546.788} C_VEL
LIN {X 0,Y 158.776,Z 329.441,A -85,B 0,C 180,E1 -23548.292,E2 -23548.292} C_VEL
LIN {X 0,Y 157.481,Z 326.769,A -85,B 0,C 180,E1 -23549.287,E2 -23549.287} C_VEL
LIN {X 0,Y 157.308,Z 325.878,A -85,B 0,C 180,E1 -23549.528,E2 -23549.528} C_VEL
LIN {X 0,Y 157.302,Z 325.882,A -85,B 0,C 180,E1 -23553.463,E2 -23553.463} C_VEL
LIN {X 0,Y 157.352,Z 325.85,A -85,B 0,C 180,E1 -23559.701,E2 -23559.701} C_VEL
LIN {X 0,Y 157.409,Z 325.828,A -85,B 0,C 180,E1 -23564.461,E2 -23564.461} C_VEL
LIN {X 0,Y 157.679,Z 325.832,A -85,B 0,C 180,E1 -23569.73,E2 -23569.73} C_VEL
LIN {X 0,Y 157.75,Z 325.778,A -85,B 0,C 180,E1 -23572.319,E2 -23572.319} C_VEL
LIN {X 0,Y 158.227,Z 325.773,A -85,B 0,C 180,E1 -23580,E2 -23580} C_VEL
LIN {X 0,Y 157.749,Z 325.83,A -85,B 0,C 180,E1 -23587.681,E2 -23587.681} C_VEL
LIN {X 0,Y 157.625,Z 325.841,A -85,B 0,C 180,E1 -23591.228,E2 -23591.228} C_VEL
LIN {X 0,Y 157.414,Z 325.852,A -85,B 0,C 180,E1 -23595.538,E2 -23595.538} C_VEL
LIN {X 0,Y 157.35,Z 325.886,A -85,B 0,C 180,E1 -23600.936,E2 -23600.936} C_VEL
LIN {X 0,Y 157.303,Z 325.872,A -85,B 0,C 180,E1 -23606.682,E2 -23606.682} C_VEL
LIN {X 0,Y 157.336,Z 325.866,A -85,B 0,C 180,E1 -23610.951,E2 -23610.951} C_VEL
LIN {X 0,Y 158.1,Z 328.428,A -85,B 0,C 180,E1 -23611.669,E2 -23611.669} C_VEL
LIN {X 0,Y 159.977,Z 330.643,A -85,B 0,C 180,E1 -23612.933,E2 -23612.933} C_VEL
LIN {X 0,Y 161.428,Z 331.722,A -85,B 0,C 180,E1 -23613.811,E2 -23613.811} C_VEL
LIN {X 0,Y 163.333,Z 334.869,A -85,B 0,C 180,E1 -23615.042,E2 -23615.042} C_VEL
LIN {X 0,Y 165.335,Z 336.969,A -85,B 0,C 180,E1 -23616.18,E2 -23616.18} C_VEL
LIN {X 0,Y 167.941,Z 340.608,A -85,B 0,C 180,E1 -23617.641,E2 -23617.641} C_VEL
LIN {X 0,Y 172.404,Z 346.924,A -85,B 0,C 180,E1 -23619.945,E2 -23619.945} C_VEL
LIN {X 0,Y 177.457,Z 354.49,A -85,B 0,C 180,E1 -23622.32,E2 -23622.32} C_VEL
LIN {X 0,Y 182.956,Z 363.535,A -85,B 0,C 180,E1 -23624.692,E2 -23624.692} C_VEL
LIN {X 0,Y 188.471,Z 373.87,A -85,B 0,C 180,E1 -23626.91,E2 -23626.91} C_VEL
LIN {X 0,Y 190.813,Z 378.719,A -85,B 0,C 180,E1 -23627.812,E2 -23627.812} C_VEL
LIN {X 0,Y 188.033,Z 424.573,A -85,B 0,C 180,E1 -23629.441,E2 -23629.441} C_VEL
LIN {X 0,Y 186.417,Z 437.901,A -85,B 0,C 180,E1 -23630.319,E2 -23630.319} C_VEL
LIN {X 0,Y 184.182,Z 450.164,A -85,B 0,C 180,E1 -23631.508,E2 -23631.508} C_VEL
LIN {X 0,Y 181.426,Z 462.009,A -85,B 0,C 180,E1 -23633.102,E2 -23633.102} C_VEL
LIN {X 0,Y 178.006,Z 473.255,A -85,B 0,C 180,E1 -23635.079,E2 -23635.079} C_VEL
LIN {X 0,Y 174.533,Z 483.4,A -85,B 0,C 180,E1 -23637.416,E2 -23637.416} C_VEL
LIN {X 0,Y 170.745,Z 493.326,A -85,B 0,C 180,E1 -23640.404,E2 -23640.404} C_VEL
LIN {X 0,Y 166.849,Z 502.003,A -85,B 0,C 180,E1 -23643.753,E2 -23643.753} C_VEL
LIN {X 0,Y 163.513,Z 508.966,A -85,B 0,C 180,E1 -23647.245,E2 -23647.245} C_VEL
LIN {X 0,Y 160.754,Z 514.492,A -85,B 0,C 180,E1 -23650.862,E2 -23650.862} C_VEL
LIN {X 0,Y 158.544,Z 518.82,A -85,B 0,C 180,E1 -23654.578,E2 -23654.578} C_VEL
LIN {X 0,Y 157.425,Z 521.092,A -85,B 0,C 180,E1 -23657.105,E2 -23657.105} C_VEL
LIN {X 0,Y 156.557,Z 522.943,A -85,B 0,C 180,E1 -23659.658,E2 -23659.658} C_VEL
LIN {X 0,Y 155.562,Z 524.969,A -85,B 0,C 180,E1 -23663.68,E2 -23663.68} C_VEL
LIN {X 0,Y 155.175,Z 525.947,A -85,B 0,C 180,E1 -23667.407,E2 -23667.407} C_VEL
LIN {X 0,Y 155.115,Z 526.175,A -85,B 0,C 180,E1 -23670.003,E2 -23670.003} C_VEL
LIN {X 0,Y 155.175,Z 525.978,A -85,B 0,C 180,E1 -23672.598,E2 -23672.598} C_VEL
LIN {X 0,Y 155.86,Z 524.425,A -85,B 0,C 180,E1 -23677.777,E2 -23677.777} C_VEL
LIN {X 0,Y 156.526,Z 523.057,A -85,B 0,C 180,E1 -23680.349,E2 -23680.349} C_VEL
LIN {X 0,Y 157.91,Z 520.185,A -85,B 0,C 180,E1 -23684.172,E2 -23684.172} C_VEL
LIN {X 0,Y 159.899,Z 516.271,A -85,B 0,C 180,E1 -23687.921,E2 -23687.921} C_VEL
LIN {X 0,Y 162.513,Z 511.196,A -85,B 0,C 180,E1 -23691.569,E2 -23691.569} C_VEL
LIN {X 0,Y 165.581,Z 504.8,A -85,B 0,C 180,E1 -23695.118,E2 -23695.118} C_VEL
LIN {X 0,Y 169.384,Z 496.822,A -85,B 0,C 180,E1 -23698.502,E2 -23698.502} C_VEL
LIN {X 0,Y 172.782,Z 488.437,A -85,B 0,C 180,E1 -23701.329,E2 -23701.329} C_VEL
LIN {X 0,Y 176.351,Z 478.604,A -85,B 0,C 180,E1 -23703.915,E2 -23703.915} C_VEL
LIN {X 0,Y 179.617,Z 468.66,A -85,B 0,C 180,E1 -23705.941,E2 -23705.941} C_VEL
LIN {X 0,Y 182.622,Z 457.822,A -85,B 0,C 180,E1 -23707.659,E2 -23707.659} C_VEL
LIN {X 0,Y 185.221,Z 445.783,A -85,B 0,C 180,E1 -23709.113,E2 -23709.113} C_VEL
LIN {X 0,Y 187.341,Z 432.396,A -85,B 0,C 180,E1 -23710.234,E2 -23710.234} C_VEL
LIN {X 0,Y 188.646,Z 419.725,A -85,B 0,C 180,E1 -23710.901,E2 -23710.901} C_VEL
LIN {X 0,Y 190.986,Z 378.959,A -85,B 0,C 180,E1 -23712.315,E2 -23712.315} C_VEL
LIN {X 0,Y 185.406,Z 367.77,A -85,B 0,C 180,E1 -23714.511,E2 -23714.511} C_VEL
LIN {X 0,Y 179.419,Z 357.445,A -85,B 0,C 180,E1 -23717.028,E2 -23717.028} C_VEL
LIN {X 0,Y 173.427,Z 348.268,A -85,B 0,C 180,E1 -23719.788,E2 -23719.788} C_VEL
LIN {X 0,Y 170.78,Z 344.533,A -85,B 0,C 180,E1 -23721.102,E2 -23721.102} C_VEL
LIN {X 0,Y 167.885,Z 340.539,A -85,B 0,C 180,E1 -23722.628,E2 -23722.628} C_VEL
LIN {X 0,Y 165.349,Z 336.938,A -85,B 0,C 180,E1 -23724.064,E2 -23724.064} C_VEL
LIN {X 0,Y 162.226,Z 333.268,A -85,B 0,C 180,E1 -23725.911,E2 -23725.911} C_VEL
LIN {X 0,Y 161.203,Z 331.391,A -85,B 0,C 180,E1 -23726.604,E2 -23726.604} C_VEL
LIN {X 0,Y 158.812,Z 329.456,A -85,B 0,C 180,E1 -23728.109,E2 -23728.109} C_VEL
LIN {X 0,Y 157.588,Z 326.993,A -85,B 0,C 180,E1 -23729.051,E2 -23729.051} C_VEL
LIN {X 0,Y 157.35,Z 325.863,A -85,B 0,C 180,E1 -23729.372,E2 -23729.372} C_VEL
LIN {X 0,Y 157.551,Z 325.945,A -85,B 0,C 180,E1 -23732.037,E2 -23732.037} C_VEL
LIN {X 0,Y 160.785,Z 339.955,A -85,B 0,C 180,E1 -23733.28,E2 -23733.28} C_VEL
LIN {X 0,Y 164.288,Z 353.411,A -85,B 0,C 180,E1 -23734.447,E2 -23734.447} C_VEL
LIN {X 0,Y 160.868,Z 425.054,A -85,B 0,C 180,E1 -23740.542,E2 -23740.542} C_VEL
LIN {X 0,Y 159.91,Z 440.312,A -85,B 0,C 180,E1 -23742.413,E2 -23742.413} C_VEL
LIN {X 0,Y 159.028,Z 453.62,A -85,B 0,C 180,E1 -23744.623,E2 -23744.623} C_VEL
LIN {X 0,Y 158.07,Z 465.676,A -85,B 0,C 180,E1 -23747.155,E2 -23747.155} C_VEL
LIN {X 0,Y 157.296,Z 476.6,A -85,B 0,C 180,E1 -23750.002,E2 -23750.002} C_VEL
LIN {X 0,Y 156.766,Z 485.873,A -85,B 0,C 180,E1 -23752.918,E2 -23752.918} C_VEL
LIN {X 0,Y 156.308,Z 494.393,A -85,B 0,C 180,E1 -23756.133,E2 -23756.133} C_VEL
LIN {X 0,Y 156.175,Z 501.553,A -85,B 0,C 180,E1 -23759.355,E2 -23759.355} C_VEL
LIN {X 0,Y 156.096,Z 508.639,A -85,B 0,C 180,E1 -23763.226,E2 -23763.226} C_VEL
LIN {X 0,Y 156.572,Z 515.345,A -85,B 0,C 180,E1 -23767.739,E2 -23767.739} C_VEL
LIN {X 0,Y 158.207,Z 521.286,A -85,B 0,C 180,E1 -23772.833,E2 -23772.833} C_VEL
LIN {X 0,Y 161.333,Z 525.744,A -85,B 0,C 180,E1 -23777.754,E2 -23777.754} C_VEL
LIN {X 0,Y 165.619,Z 528.818,A -85,B 0,C 180,E1 -23782.452,E2 -23782.452} C_VEL
LIN {X 0,Y 171.41,Z 530.575,A -85,B 0,C 180,E1 -23786.809,E2 -23786.809} C_VEL
LIN {X 0,Y 178.387,Z 531.011,A -85,B 0,C 180,E1 -23790.808,E2 -23790.808} C_VEL
LIN {X 0,Y 186.487,Z 530.149,A -85,B 0,C 180,E1 -23794.423,E2 -23794.423} C_VEL
LIN {X 0,Y 195.544,Z 527.968,A -85,B 0,C 180,E1 -23797.661,E2 -23797.661} C_VEL
LIN {X 0,Y 205.442,Z 524.388,A -85,B 0,C 180,E1 -23800.54,E2 -23800.54} C_VEL
LIN {X 0,Y 216.04,Z 519.285,A -85,B 0,C 180,E1 -23803.09,E2 -23803.09} C_VEL
LIN {X 0,Y 218.324,Z 518.057,A -85,B 0,C 180,E1 -23803.575,E2 -23803.575} C_VEL
LIN {X 0,Y 217.709,Z 518.518,A -85,B 0,C 180,E1 -23804.114,E2 -23804.114} C_VEL
LIN {X 0,Y 207.976,Z 524.243,A -85,B 0,C 180,E1 -23806.15,E2 -23806.15} C_VEL
LIN {X 0,Y 197.574,Z 529.379,A -85,B 0,C 180,E1 -23808.845,E2 -23808.845} C_VEL
LIN {X 0,Y 190.355,Z 532.352,A -85,B 0,C 180,E1 -23811.121,E2 -23811.121} C_VEL
LIN {X 0,Y 181.48,Z 535.16,A -85,B 0,C 180,E1 -23814.484,E2 -23814.484} C_VEL
LIN {X 0,Y 173.784,Z 536.744,A -85,B 0,C 180,E1 -23818.28,E2 -23818.28} C_VEL
LIN {X 0,Y 172.682,Z 536.863,A -85,B 0,C 180,E1 -23818.96,E2 -23818.96} C_VEL
LIN {X 0,Y 169.44,Z 537.104,A -85,B 0,C 180,E1 -23820.613,E2 -23820.613} C_VEL
LIN {X 0,Y 162.927,Z 536.672,A -85,B 0,C 180,E1 -23823.184,E2 -23823.184} C_VEL
LIN {X 0,Y 156.898,Z 535.466,A -85,B 0,C 180,E1 -23825.969,E2 -23825.969} C_VEL
LIN {X 0,Y 154.498,Z 534.488,A -85,B 0,C 180,E1 -23827.927,E2 -23827.927} C_VEL
LIN {X 0,Y 151.43,Z 531.744,A -85,B 0,C 180,E1 -23833.309,E2 -23833.309} C_VEL
LIN {X 0,Y 149.763,Z 534.527,A -85,B 0,C 180,E1 -23836.427,E2 -23836.427} C_VEL
LIN {X 0,Y 148.815,Z 536.42,A -85,B 0,C 180,E1 -23839.108,E2 -23839.108} C_VEL
LIN {X 0,Y 148.217,Z 537.85,A -85,B 0,C 180,E1 -23841.819,E2 -23841.819} C_VEL
LIN {X 0,Y 147.861,Z 539.354,A -85,B 0,C 180,E1 -23846.521,E2 -23846.521} C_VEL
LIN {X 0,Y 148.053,Z 539.718,A -85,B 0,C 180,E1 -23849.997,E2 -23849.997} C_VEL
LIN {X 0,Y 147.814,Z 539.394,A -85,B 0,C 180,E1 -23853.167,E2 -23853.167} C_VEL
LIN {X 0,Y 147.885,Z 537.8,A -85,B 0,C 180,E1 -23858.194,E2 -23858.194} C_VEL
LIN {X 0,Y 148.277,Z 536.341,A -85,B 0,C 180,E1 -23860.926,E2 -23860.926} C_VEL
LIN {X 0,Y 149.35,Z 533.326,A -85,B 0,C 180,E1 -23864.997,E2 -23864.997} C_VEL
LIN {X 0,Y 151.234,Z 529.258,A -85,B 0,C 180,E1 -23868.981,E2 -23868.981} C_VEL
LIN {X 0,Y 154.378,Z 523.003,A -85,B 0,C 180,E1 -23873.471,E2 -23873.471} C_VEL
LIN {X 0,Y 157.571,Z 516.182,A -85,B 0,C 180,E1 -23877.202,E2 -23877.202} C_VEL
LIN {X 0,Y 160.765,Z 509.225,A -85,B 0,C 180,E1 -23880.178,E2 -23880.178} C_VEL
LIN {X 0,Y 164.484,Z 500.839,A -85,B 0,C 180,E1 -23883.006,E2 -23883.006} C_VEL
LIN {X 0,Y 168.67,Z 490.468,A -85,B 0,C 180,E1 -23885.683,E2 -23885.683} C_VEL
LIN {X 0,Y 172.74,Z 478.8,A -85,B 0,C 180,E1 -23887.975,E2 -23887.975} C_VEL
LIN {X 0,Y 176.112,Z 467.055,A -85,B 0,C 180,E1 -23889.677,E2 -23889.677} C_VEL
LIN {X 0,Y 178.916,Z 454.901,A -85,B 0,C 180,E1 -23890.954,E2 -23890.954} C_VEL
LIN {X 0,Y 181.032,Z 442.558,A -85,B 0,C 180,E1 -23891.844,E2 -23891.844} C_VEL
LIN {X 0,Y 182.29,Z 428.674,A -85,B 0,C 180,E1 -23892.483,E2 -23892.483} C_VEL
LIN {X 0,Y 184.244,Z 395.499,A -85,B 0,C 180,E1 -23893.65,E2 -23893.65} C_VEL
LIN {X 0,Y 182.88,Z 377.359,A -85,B 0,C 180,E1 -23895.029,E2 -23895.029} C_VEL
LIN {X 0,Y 181.482,Z 372.959,A -85,B 0,C 180,E1 -23895.711,E2 -23895.711} C_VEL
LIN {X 0,Y 175.003,Z 361.547,A -85,B 0,C 180,E1 -23898.597,E2 -23898.597} C_VEL
LIN {X 0,Y 169.111,Z 352.446,A -85,B 0,C 180,E1 -23901.496,E2 -23901.496} C_VEL
LIN {X 0,Y 164.566,Z 346.004,A -85,B 0,C 180,E1 -23903.976,E2 -23903.976} C_VEL
LIN {X 0,Y 161.701,Z 341.994,A -85,B 0,C 180,E1 -23905.691,E2 -23905.691} C_VEL
LIN {X 0,Y 159.12,Z 338.631,A -85,B 0,C 180,E1 -23907.338,E2 -23907.338} C_VEL
LIN {X 0,Y 158.404,Z 337.539,A -85,B 0,C 180,E1 -23907.832,E2 -23907.832} C_VEL
LIN {X 0,Y 156.006,Z 335.157,A -85,B 0,C 180,E1 -23909.457,E2 -23909.457} C_VEL
LIN {X 0,Y 154.426,Z 332.406,A -85,B 0,C 180,E1 -23910.709,E2 -23910.709} C_VEL
LIN {X 0,Y 151.968,Z 330.647,A -85,B 0,C 180,E1 -23912.565,E2 -23912.565} C_VEL
LIN {X 0,Y 150.515,Z 328.028,A -85,B 0,C 180,E1 -23913.914,E2 -23913.914} C_VEL
LIN {X 0,Y 150.223,Z 326.76,A -85,B 0,C 180,E1 -23914.318,E2 -23914.318} C_VEL
LIN {X 0,Y 150.276,Z 326.736,A -85,B 0,C 180,E1 -23919.276,E2 -23919.276} C_VEL
LIN {X 0,Y 150.312,Z 326.703,A -85,B 0,C 180,E1 -23923.708,E2 -23923.708} C_VEL
LIN {X 0,Y 150.6,Z 326.719,A -85,B 0,C 180,E1 -23929.242,E2 -23929.242} C_VEL
LIN {X 0,Y 150.673,Z 326.661,A -85,B 0,C 180,E1 -23931.956,E2 -23931.956} C_VEL
LIN {X 0,Y 151.188,Z 326.65,A -85,B 0,C 180,E1 -23940,E2 -23940} C_VEL
LIN {X 0,Y 150.672,Z 326.707,A -85,B 0,C 180,E1 -23948.044,E2 -23948.044} C_VEL
LIN {X 0,Y 150.566,Z 326.721,A -85,B 0,C 180,E1 -23951.431,E2 -23951.431} C_VEL
LIN {X 0,Y 150.321,Z 326.729,A -85,B 0,C 180,E1 -23956.291,E2 -23956.291} C_VEL
LIN {X 0,Y 150.332,Z 326.759,A -85,B 0,C 180,E1 -23960.781,E2 -23960.781} C_VEL
LIN {X 0,Y 150.264,Z 326.852,A -85,B 0,C 180,E1 -23966.208,E2 -23966.208} C_VEL
LIN {X 0,Y 151.149,Z 329.483,A -85,B 0,C 180,E1 -23967.16,E2 -23967.16} C_VEL
LIN {X 0,Y 153.144,Z 331.7,A -85,B 0,C 180,E1 -23968.807,E2 -23968.807} C_VEL
LIN {X 0,Y 154.742,Z 332.771,A -85,B 0,C 180,E1 -23969.973,E2 -23969.973} C_VEL
LIN {X 0,Y 156.388,Z 335.697,A -85,B 0,C 180,E1 -23971.269,E2 -23971.269} C_VEL
LIN {X 0,Y 158.844,Z 338.174,A -85,B 0,C 180,E1 -23972.914,E2 -23972.914} C_VEL
LIN {X 0,Y 161.28,Z 341.614,A -85,B 0,C 180,E1 -23974.506,E2 -23974.506} C_VEL
LIN {X 0,Y 162.712,Z 343.405,A -85,B 0,C 180,E1 -23975.374,E2 -23975.374} C_VEL
LIN {X 0,Y 166.178,Z 348.252,A -85,B 0,C 180,E1 -23977.379,E2 -23977.379} C_VEL
LIN {X 0,Y 171.353,Z 355.839,A -85,B 0,C 180,E1 -23980.096,E2 -23980.096} C_VEL
LIN {X 0,Y 177.344,Z 365.556,A -85,B 0,C 180,E1 -23982.932,E2 -23982.932} C_VEL
LIN {X 0,Y 182.487,Z 375.016,A -85,B 0,C 180,E1 -23985.173,E2 -23985.173} C_VEL
LIN {X 0,Y 185.521,Z 381.33,A -85,B 0,C 180,E1 -23986.438,E2 -23986.438} C_VEL
LIN {X 0,Y 182.71,Z 424.834,A -85,B 0,C 180,E1 -23987.996,E2 -23987.996} C_VEL
LIN {X 0,Y 181.027,Z 438.19,A -85,B 0,C 180,E1 -23988.889,E2 -23988.889} C_VEL
LIN {X 0,Y 178.683,Z 450.464,A -85,B 0,C 180,E1 -23990.091,E2 -23990.091} C_VEL
LIN {X 0,Y 175.817,Z 462.315,A -85,B 0,C 180,E1 -23991.717,E2 -23991.717} C_VEL
LIN {X 0,Y 172.231,Z 473.566,A -85,B 0,C 180,E1 -23993.727,E2 -23993.727} C_VEL
LIN {X 0,Y 168.59,Z 483.713,A -85,B 0,C 180,E1 -23996.116,E2 -23996.116} C_VEL
LIN {X 0,Y 165.44,Z 491.894,A -85,B 0,C 180,E1 -23998.598,E2 -23998.598} C_VEL
LIN {X 0,Y 161.855,Z 499.659,A -85,B 0,C 180,E1 -24001.472,E2 -24001.472} C_VEL
LIN {X 0,Y 158.093,Z 507.114,A -85,B 0,C 180,E1 -24005.022,E2 -24005.022} C_VEL
LIN {X 0,Y 155.005,Z 513.089,A -85,B 0,C 180,E1 -24008.735,E2 -24008.735} C_VEL
LIN {X 0,Y 152.451,Z 517.809,A -85,B 0,C 180,E1 -24012.566,E2 -24012.566} C_VEL
LIN {X 0,Y 150.53,Z 521.409,A -85,B 0,C 180,E1 -24016.503,E2 -24016.503} C_VEL
LIN {X 0,Y 149.586,Z 523.26,A -85,B 0,C 180,E1 -24019.171,E2 -24019.171} C_VEL
LIN {X 0,Y 148.468,Z 525.425,A -85,B 0,C 180,E1 -24023.76,E2 -24023.76} C_VEL
LIN {X 0,Y 148.092,Z 526.264,A -85,B 0,C 180,E1 -24027.283,E2 -24027.283} C_VEL
LIN {X 0,Y 148.024,Z 526.491,A -85,B 0,C 180,E1 -24030.003,E2 -24030.003} C_VEL
LIN {X 0,Y 148.092,Z 526.294,A -85,B 0,C 180,E1 -24032.723,E2 -24032.723} C_VEL
LIN {X 0,Y 148.839,Z 524.741,A -85,B 0,C 180,E1 -24038.146,E2 -24038.146} C_VEL
LIN {X 0,Y 149.563,Z 523.372,A -85,B 0,C 180,E1 -24040.836,E2 -24040.836} C_VEL
LIN {X 0,Y 151.034,Z 520.5,A -85,B 0,C 180,E1 -24044.831,E2 -24044.831} C_VEL
LIN {X 0,Y 153.172,Z 516.585,A -85,B 0,C 180,E1 -24048.737,E2 -24048.737} C_VEL
LIN {X 0,Y 155.916,Z 511.51,A -85,B 0,C 180,E1 -24052.531,E2 -24052.531} C_VEL
LIN {X 0,Y 159.203,Z 505.111,A -85,B 0,C 180,E1 -24056.199,E2 -24056.199} C_VEL
LIN {X 0,Y 163.201,Z 497.131,A -85,B 0,C 180,E1 -24059.688,E2 -24059.688} C_VEL
LIN {X 0,Y 166.567,Z 489.212,A -85,B 0,C 180,E1 -24062.449,E2 -24062.449} C_VEL
LIN {X 0,Y 170.121,Z 480.045,A -85,B 0,C 180,E1 -24064.976,E2 -24064.976} C_VEL
LIN {X 0,Y 173.932,Z 468.96,A -85,B 0,C 180,E1 -24067.311,E2 -24067.311} C_VEL
LIN {X 0,Y 177.068,Z 458.116,A -85,B 0,C 180,E1 -24069.06,E2 -24069.06} C_VEL
LIN {X 0,Y 179.788,Z 446.063,A -85,B 0,C 180,E1 -24070.535,E2 -24070.535} C_VEL
LIN {X 0,Y 181.933,Z 433.143,A -85,B 0,C 180,E1 -24071.638,E2 -24071.638} C_VEL
LIN {X 0,Y 183.343,Z 419.909,A -85,B 0,C 180,E1 -24072.354,E2 -24072.354} C_VEL
LIN {X 0,Y 185.654,Z 381.428,A -85,B 0,C 180,E1 -24073.711,E2 -24073.711} C_VEL
LIN {X 0,Y 180.268,Z 370.563,A -85,B 0,C 180,E1 -24075.992,E2 -24075.992} C_VEL
LIN {X 0,Y 174.326,Z 360.383,A -85,B 0,C 180,E1 -24078.687,E2 -24078.687} C_VEL
LIN {X 0,Y 168.219,Z 350.924,A -85,B 0,C 180,E1 -24081.767,E2 -24081.767} C_VEL
LIN {X 0,Y 164.63,Z 346.015,A -85,B 0,C 180,E1 -24083.748,E2 -24083.748} C_VEL
LIN {X 0,Y 161.723,Z 342.005,A -85,B 0,C 180,E1 -24085.496,E2 -24085.496} C_VEL
LIN {X 0,Y 159.201,Z 338.729,A -85,B 0,C 180,E1 -24087.116,E2 -24087.116} C_VEL
LIN {X 0,Y 158.432,Z 337.551,A -85,B 0,C 180,E1 -24087.649,E2 -24087.649} C_VEL
LIN {X 0,Y 155.934,Z 335.001,A -85,B 0,C 180,E1 -24089.366,E2 -24089.366} C_VEL
LIN {X 0,Y 155.036,Z 333.314,A -85,B 0,C 180,E1 -24090.089,E2 -24090.089} C_VEL
LIN {X 0,Y 154.027,Z 333.667,A -85,B 0,C 180,E1 -24090.72,E2 -24090.72} C_VEL
LIN {X 0,Y 153.205,Z 334.408,A -85,B 0,C 180,E1 -24091.205,E2 -24091.205} C_VEL
LIN {X 0,Y 152.148,Z 334.013,A -85,B 0,C 180,E1 -24091.983,E2 -24091.983} C_VEL
LIN {X 0,Y 151.665,Z 332.758,A -85,B 0,C 180,E1 -24092.456,E2 -24092.456} C_VEL
LIN {X 0,Y 157.111,Z 354.502,A -85,B 0,C 180,E1 -24094.467,E2 -24094.467} C_VEL
LIN {X 0,Y 153.78,Z 425.037,A -85,B 0,C 180,E1 -24100.823,E2 -24100.823} C_VEL
LIN {X 0,Y 152.855,Z 440.262,A -85,B 0,C 180,E1 -24102.783,E2 -24102.783} C_VEL
LIN {X 0,Y 152.054,Z 452.738,A -85,B 0,C 180,E1 -24104.93,E2 -24104.93} C_VEL
LIN {X 0,Y 151.094,Z 465.17,A -85,B 0,C 180,E1 -24107.644,E2 -24107.644} C_VEL
LIN {X 0,Y 150.324,Z 476.474,A -85,B 0,C 180,E1 -24110.709,E2 -24110.709} C_VEL
LIN {X 0,Y 149.825,Z 486.228,A -85,B 0,C 180,E1 -24113.941,E2 -24113.941} C_VEL
LIN {X 0,Y 149.414,Z 496.208,A -85,B 0,C 180,E1 -24117.978,E2 -24117.978} C_VEL
LIN {X 0,Y 149.255,Z 503.003,A -85,B 0,C 180,E1 -24121.349,E2 -24121.349} C_VEL
LIN {X 0,Y 149.427,Z 509.826,A -85,B 0,C 180,E1 -24125.397,E2 -24125.397} C_VEL
LIN {X 0,Y 149.954,Z 515.086,A -85,B 0,C 180,E1 -24129.185,E2 -24129.185} C_VEL
LIN {X 0,Y 152.087,Z 521.422,A -85,B 0,C 180,E1 -24134.724,E2 -24134.724} C_VEL
LIN {X 0,Y 154.634,Z 524.957,A -85,B 0,C 180,E1 -24138.551,E2 -24138.551} C_VEL
LIN {X 0,Y 159.107,Z 528.437,A -85,B 0,C 180,E1 -24143.425,E2 -24143.425} C_VEL
LIN {X 0,Y 165.118,Z 530.63,A -85,B 0,C 180,E1 -24147.917,E2 -24147.917} C_VEL
LIN {X 0,Y 172.356,Z 531.559,A -85,B 0,C 180,E1 -24152.011,E2 -24152.011} C_VEL
LIN {X 0,Y 180.733,Z 531.215,A -85,B 0,C 180,E1 -24155.682,E2 -24155.682} C_VEL
LIN {X 0,Y 190.09,Z 529.589,A -85,B 0,C 180,E1 -24158.941,E2 -24158.941} C_VEL
LIN {X 0,Y 200.282,Z 526.597,A -85,B 0,C 180,E1 -24161.814,E2 -24161.814} C_VEL
LIN {X 0,Y 206.75,Z 524.101,A -85,B 0,C 180,E1 -24163.375,E2 -24163.375} C_VEL
LIN {X 0,Y 206.865,Z 524.157,A -85,B 0,C 180,E1 -24163.948,E2 -24163.948} C_VEL
LIN {X 0,Y 197.559,Z 528.459,A -85,B 0,C 180,E1 -24166.074,E2 -24166.074} C_VEL
LIN {X 0,Y 189.805,Z 531.476,A -85,B 0,C 180,E1 -24168.2,E2 -24168.2} C_VEL
LIN {X 0,Y 180.217,Z 534.372,A -85,B 0,C 180,E1 -24171.392,E2 -24171.392} C_VEL
LIN {X 0,Y 171.635,Z 536.056,A -85,B 0,C 180,E1 -24175.019,E2 -24175.019} C_VEL
LIN {X 0,Y 164.414,Z 536.591,A -85,B 0,C 180,E1 -24179.137,E2 -24179.137} C_VEL
LIN {X 0,Y 158.505,Z 535.986,A -85,B 0,C 180,E1 -24183.677,E2 -24183.677} C_VEL
LIN {X 0,Y 154.498,Z 534.488,A -85,B 0,C 180,E1 -24187.927,E2 -24187.927} C_VEL
LIN {X 0,Y 152.802,Z 533.83,A -85,B 0,C 180,E1 -24189.279,E2 -24189.279} C_VEL
LIN {X 0,Y 148.622,Z 532.844,A -85,B 0,C 180,E1 -24191.31,E2 -24191.31} C_VEL
LIN {X 0,Y 145.317,Z 532.669,A -85,B 0,C 180,E1 -24192.982,E2 -24192.982} C_VEL
LIN {X 0,Y 143.482,Z 533.266,A -85,B 0,C 180,E1 -24194.51,E2 -24194.51} C_VEL
LIN {X 0,Y 143.26,Z 533.531,A -85,B 0,C 180,E1 -24194.883,E2 -24194.883} C_VEL
LIN {X 0,Y 141.845,Z 536.104,A -85,B 0,C 180,E1 -24198.566,E2 -24198.566} C_VEL
LIN {X 0,Y 141.173,Z 537.533,A -85,B 0,C 180,E1 -24201.408,E2 -24201.408} C_VEL
LIN {X 0,Y 140.778,Z 539.119,A -85,B 0,C 180,E1 -24206.814,E2 -24206.814} C_VEL
LIN {X 0,Y 140.952,Z 539.401,A -85,B 0,C 180,E1 -24209.997,E2 -24209.997} C_VEL
LIN {X 0,Y 140.735,Z 539.157,A -85,B 0,C 180,E1 -24212.86,E2 -24212.86} C_VEL
LIN {X 0,Y 140.829,Z 537.482,A -85,B 0,C 180,E1 -24218.607,E2 -24218.607} C_VEL
LIN {X 0,Y 141.275,Z 536.021,A -85,B 0,C 180,E1 -24221.475,E2 -24221.475} C_VEL
LIN {X 0,Y 142.446,Z 533.006,A -85,B 0,C 180,E1 -24225.742,E2 -24225.742} C_VEL
LIN {X 0,Y 144.51,Z 528.94,A -85,B 0,C 180,E1 -24229.9,E2 -24229.9} C_VEL
LIN {X 0,Y 147.875,Z 522.686,A -85,B 0,C 180,E1 -24234.57,E2 -24234.57} C_VEL
LIN {X 0,Y 151.251,Z 515.864,A -85,B 0,C 180,E1 -24238.439,E2 -24238.439} C_VEL
LIN {X 0,Y 154.637,Z 508.908,A -85,B 0,C 180,E1 -24241.507,E2 -24241.507} C_VEL
LIN {X 0,Y 158.551,Z 500.524,A -85,B 0,C 180,E1 -24244.41,E2 -24244.41} C_VEL
LIN {X 0,Y 162.945,Z 490.156,A -85,B 0,C 180,E1 -24247.142,E2 -24247.142} C_VEL
LIN {X 0,Y 167.183,Z 478.491,A -85,B 0,C 180,E1 -24249.477,E2 -24249.477} C_VEL
LIN {X 0,Y 170.713,Z 466.752,A -85,B 0,C 180,E1 -24251.197,E2 -24251.197} C_VEL
LIN {X 0,Y 173.621,Z 454.606,A -85,B 0,C 180,E1 -24252.489,E2 -24252.489} C_VEL
LIN {X 0,Y 175.897,Z 441.643,A -85,B 0,C 180,E1 -24253.421,E2 -24253.421} C_VEL
LIN {X 0,Y 177.2,Z 426.956,A -85,B 0,C 180,E1 -24254.091,E2 -24254.091} C_VEL
LIN {X 0,Y 179.075,Z 396.095,A -85,B 0,C 180,E1 -24255.203,E2 -24255.203} C_VEL
LIN {X 0,Y 177.975,Z 379.853,A -85,B 0,C 180,E1 -24256.477,E2 -24256.477} C_VEL
LIN {X 0,Y 177.019,Z 376.963,A -85,B 0,C 180,E1 -24256.968,E2 -24256.968} C_VEL
LIN {X 0,Y 171.102,Z 366.328,A -85,B 0,C 180,E1 -24259.786,E2 -24259.786} C_VEL
LIN {X 0,Y 164.775,Z 356.28,A -85,B 0,C 180,E1 -24263.145,E2 -24263.145} C_VEL
LIN {X 0,Y 158.998,Z 348.007,A -85,B 0,C 180,E1 -24266.65,E2 -24266.65} C_VEL
LIN {X 0,Y 156.317,Z 344.379,A -85,B 0,C 180,E1 -24268.47,E2 -24268.47} C_VEL
LIN {X 0,Y 153.065,Z 340.478,A -85,B 0,C 180,E1 -24270.857,E2 -24270.857} C_VEL
LIN {X 0,Y 152.279,Z 338.96,A -85,B 0,C 180,E1 -24271.532,E2 -24271.532} C_VEL
LIN {X 0,Y 149.63,Z 336.699,A -85,B 0,C 180,E1 -24273.682,E2 -24273.682} C_VEL
LIN {X 0,Y 147.888,Z 333.483,A -85,B 0,C 180,E1 -24275.429,E2 -24275.429} C_VEL
LIN {X 0,Y 145.346,Z 331.937,A -85,B 0,C 180,E1 -24277.892,E2 -24277.892} C_VEL
LIN {X 0,Y 143.714,Z 329.422,A -85,B 0,C 180,E1 -24279.886,E2 -24279.886} C_VEL
LIN {X 0,Y 143.254,Z 327.586,A -85,B 0,C 180,E1 -24280.754,E2 -24280.754} C_VEL
LIN {X 0,Y 143.526,Z 327.604,A -85,B 0,C 180,E1 -24288.705,E2 -24288.705} C_VEL
LIN {X 0,Y 143.599,Z 327.545,A -85,B 0,C 180,E1 -24291.557,E2 -24291.557} C_VEL
LIN {X 0,Y 144.146,Z 327.527,A -85,B 0,C 180,E1 -24300,E2 -24300} C_VEL
LIN {X 0,Y 143.598,Z 327.584,A -85,B 0,C 180,E1 -24308.443,E2 -24308.443} C_VEL
LIN {X 0,Y 143.493,Z 327.603,A -85,B 0,C 180,E1 -24311.619,E2 -24311.619} C_VEL
LIN {X 0,Y 143.271,Z 327.619,A -85,B 0,C 180,E1 -24319.337,E2 -24319.337} C_VEL
LIN {X 0,Y 143.261,Z 327.644,A -85,B 0,C 180,E1 -24319.804,E2 -24319.804} C_VEL
LIN {X 0,Y 143.987,Z 329.972,A -85,B 0,C 180,E1 -24320.925,E2 -24320.925} C_VEL
LIN {X 0,Y 145.666,Z 332.228,A -85,B 0,C 180,E1 -24322.892,E2 -24322.892} C_VEL
LIN {X 0,Y 148.073,Z 333.706,A -85,B 0,C 180,E1 -24325.194,E2 -24325.194} C_VEL
LIN {X 0,Y 149.529,Z 336.564,A -85,B 0,C 180,E1 -24326.671,E2 -24326.671} C_VEL
LIN {X 0,Y 152.158,Z 338.9,A -85,B 0,C 180,E1 -24328.823,E2 -24328.823} C_VEL
LIN {X 0,Y 154.669,Z 342.614,A -85,B 0,C 180,E1 -24330.819,E2 -24330.819} C_VEL
LIN {X 0,Y 156.32,Z 344.441,A -85,B 0,C 180,E1 -24331.984,E2 -24331.984} C_VEL
LIN {X 0,Y 159.136,Z 348.209,A -85,B 0,C 180,E1 -24333.888,E2 -24333.888} C_VEL
LIN {X 0,Y 165.213,Z 356.953,A -85,B 0,C 180,E1 -24337.552,E2 -24337.552} C_VEL
LIN {X 0,Y 171.895,Z 367.684,A -85,B 0,C 180,E1 -24341.06,E2 -24341.06} C_VEL
LIN {X 0,Y 177.831,Z 378.6,A -85,B 0,C 180,E1 -24343.856,E2 -24343.856} C_VEL
LIN {X 0,Y 180.292,Z 383.776,A -85,B 0,C 180,E1 -24344.959,E2 -24344.959} C_VEL
LIN {X 0,Y 177.54,Z 424.746,A -85,B 0,C 180,E1 -24346.45,E2 -24346.45} C_VEL
LIN {X 0,Y 175.878,Z 437.761,A -85,B 0,C 180,E1 -24347.311,E2 -24347.311} C_VEL
LIN {X 0,Y 173.306,Z 450.764,A -85,B 0,C 180,E1 -24348.588,E2 -24348.588} C_VEL
LIN {X 0,Y 170.311,Z 462.621,A -85,B 0,C 180,E1 -24350.24,E2 -24350.24} C_VEL
LIN {X 0,Y 166.581,Z 473.875,A -85,B 0,C 180,E1 -24352.287,E2 -24352.287} C_VEL
LIN {X 0,Y 162.749,Z 484.025,A -85,B 0,C 180,E1 -24354.723,E2 -24354.723} C_VEL
LIN {X 0,Y 159.344,Z 492.406,A -85,B 0,C 180,E1 -24357.336,E2 -24357.336} C_VEL
LIN {X 0,Y 154.937,Z 501.311,A -85,B 0,C 180,E1 -24360.819,E2 -24360.819} C_VEL
LIN {X 0,Y 151.104,Z 508.521,A -85,B 0,C 180,E1 -24364.521,E2 -24364.521} C_VEL
LIN {X 0,Y 147.431,Z 515.126,A -85,B 0,C 180,E1 -24369.055,E2 -24369.055} C_VEL
LIN {X 0,Y 144.933,Z 519.453,A -85,B 0,C 180,E1 -24373.088,E2 -24373.088} C_VEL
LIN {X 0,Y 143.639,Z 521.726,A -85,B 0,C 180,E1 -24375.842,E2 -24375.842} C_VEL
LIN {X 0,Y 142.618,Z 523.578,A -85,B 0,C 180,E1 -24378.635,E2 -24378.635} C_VEL
LIN {X 0,Y 141.342,Z 525.887,A -85,B 0,C 180,E1 -24383.974,E2 -24383.974} C_VEL
LIN {X 0,Y 141.011,Z 526.581,A -85,B 0,C 180,E1 -24387.146,E2 -24387.146} C_VEL
LIN {X 0,Y 140.935,Z 526.808,A -85,B 0,C 180,E1 -24390.003,E2 -24390.003} C_VEL
LIN {X 0,Y 141.011,Z 526.611,A -85,B 0,C 180,E1 -24392.86,E2 -24392.86} C_VEL
LIN {X 0,Y 141.818,Z 525.058,A -85,B 0,C 180,E1 -24398.553,E2 -24398.553} C_VEL
LIN {X 0,Y 142.598,Z 523.689,A -85,B 0,C 180,E1 -24401.373,E2 -24401.373} C_VEL
LIN {X 0,Y 144.194,Z 520.815,A -85,B 0,C 180,E1 -24405.552,E2 -24405.552} C_VEL
LIN {X 0,Y 146.482,Z 516.899,A -85,B 0,C 180,E1 -24409.627,E2 -24409.627} C_VEL
LIN {X 0,Y 149.375,Z 511.824,A -85,B 0,C 180,E1 -24413.576,E2 -24413.576} C_VEL
LIN {X 0,Y 152.872,Z 505.423,A -85,B 0,C 180,E1 -24417.372,E2 -24417.372} C_VEL
LIN {X 0,Y 157.086,Z 497.441,A -85,B 0,C 180,E1 -24420.967,E2 -24420.967} C_VEL
LIN {X 0,Y 160.967,Z 488.712,A -85,B 0,C 180,E1 -24424.067,E2 -24424.067} C_VEL
LIN {X 0,Y 164.772,Z 479.212,A -85,B 0,C 180,E1 -24426.668,E2 -24426.668} C_VEL
LIN {X 0,Y 168.852,Z 467.875,A -85,B 0,C 180,E1 -24429.019,E2 -24429.019} C_VEL
LIN {X 0,Y 172.072,Z 456.646,A -85,B 0,C 180,E1 -24430.808,E2 -24430.808} C_VEL
LIN {X 0,Y 174.721,Z 445.106,A -85,B 0,C 180,E1 -24432.165,E2 -24432.165} C_VEL
LIN {X 0,Y 176.918,Z 431.798,A -85,B 0,C 180,E1 -24433.283,E2 -24433.283} C_VEL
LIN {X 0,Y 178.249,Z 418.952,A -85,B 0,C 180,E1 -24433.935,E2 -24433.935} C_VEL
LIN {X 0,Y 180.429,Z 383.855,A -85,B 0,C 180,E1 -24435.194,E2 -24435.194} C_VEL
LIN {X 0,Y 175.306,Z 373.623,A -85,B 0,C 180,E1 -24437.525,E2 -24437.525} C_VEL
LIN {X 0,Y 170.344,Z 364.995,A -85,B 0,C 180,E1 -24439.947,E2 -24439.947} C_VEL
LIN {X 0,Y 165.001,Z 356.496,A -85,B 0,C 180,E1 -24442.821,E2 -24442.821} C_VEL
LIN {X 0,Y 161.427,Z 351.482,A -85,B 0,C 180,E1 -24444.92,E2 -24444.92} C_VEL
LIN {X 0,Y 158.908,Z 347.912,A -85,B 0,C 180,E1 -24446.531,E2 -24446.531} C_VEL
LIN {X 0,Y 155.703,Z 343.604,A -85,B 0,C 180,E1 -24448.748,E2 -24448.748} C_VEL
LIN {X 0,Y 153.323,Z 341.234,A -85,B 0,C 180,E1 -24450.478,E2 -24450.478} C_VEL
LIN {X 0,Y 151.263,Z 346.579,A -85,B 0,C 180,E1 -24451.37,E2 -24451.37} C_VEL
LIN {X 0,Y 150.034,Z 348.378,A -85,B 0,C 180,E1 -24452.067,E2 -24452.067} C_VEL
LIN {X 0,Y 149.478,Z 348.793,A -85,B 0,C 180,E1 -24452.433,E2 -24452.433} C_VEL
LIN {X 0,Y 148.51,Z 348.342,A -85,B 0,C 180,E1 -24453.21,E2 -24453.21} C_VEL
LIN {X 0,Y 148.042,Z 347.149,A -85,B 0,C 180,E1 -24453.703,E2 -24453.703} C_VEL
LIN {X 0,Y 149.965,Z 355.177,A -85,B 0,C 180,E1 -24454.488,E2 -24454.488} C_VEL
LIN {X 0,Y 146.731,Z 424.718,A -85,B 0,C 180,E1 -24461.137,E2 -24461.137} C_VEL
LIN {X 0,Y 145.834,Z 439.955,A -85,B 0,C 180,E1 -24463.193,E2 -24463.193} C_VEL
LIN {X 0,Y 144.967,Z 453.328,A -85,B 0,C 180,E1 -24465.613,E2 -24465.613} C_VEL
LIN {X 0,Y 144.068,Z 465.53,A -85,B 0,C 180,E1 -24468.442,E2 -24468.442} C_VEL
LIN {X 0,Y 143.403,Z 476.376,A -85,B 0,C 180,E1 -24471.545,E2 -24471.545} C_VEL
LIN {X 0,Y 142.881,Z 486.422,A -85,B 0,C 180,E1 -24475.062,E2 -24475.062} C_VEL
LIN {X 0,Y 142.617,Z 496.338,A -85,B 0,C 180,E1 -24479.294,E2 -24479.294} C_VEL
LIN {X 0,Y 142.501,Z 504.267,A -85,B 0,C 180,E1 -24483.534,E2 -24483.534} C_VEL
LIN {X 0,Y 142.81,Z 509.814,A -85,B 0,C 180,E1 -24487.067,E2 -24487.067} C_VEL
LIN {X 0,Y 144.091,Z 517.084,A -85,B 0,C 180,E1 -24492.7,E2 -24492.7} C_VEL
LIN {X 0,Y 147.031,Z 522.739,A -85,B 0,C 180,E1 -24498.101,E2 -24498.101} C_VEL
LIN {X 0,Y 150.153,Z 526.063,A -85,B 0,C 180,E1 -24501.99,E2 -24501.99} C_VEL
LIN {X 0,Y 155.605,Z 529.336,A -85,B 0,C 180,E1 -24506.85,E2 -24506.85} C_VEL
LIN {X 0,Y 162.471,Z 531.373,A -85,B 0,C 180,E1 -24511.271,E2 -24511.271} C_VEL
LIN {X 0,Y 170.608,Z 532.168,A -85,B 0,C 180,E1 -24515.22,E2 -24515.22} C_VEL
LIN {X 0,Y 179.752,Z 531.721,A -85,B 0,C 180,E1 -24518.724,E2 -24518.724} C_VEL
LIN {X 0,Y 189.835,Z 529.985,A -85,B 0,C 180,E1 -24521.789,E2 -24521.789} C_VEL
LIN {X 0,Y 195.974,Z 528.369,A -85,B 0,C 180,E1 -24523.363,E2 -24523.363} C_VEL
LIN {X 0,Y 195.301,Z 528.715,A -85,B 0,C 180,E1 -24523.967,E2 -24523.967} C_VEL
LIN {X 0,Y 184.591,Z 532.28,A -85,B 0,C 180,E1 -24526.737,E2 -24526.737} C_VEL
LIN {X 0,Y 174.727,Z 534.629,A -85,B 0,C 180,E1 -24529.939,E2 -24529.939} C_VEL
LIN {X 0,Y 165.887,Z 535.816,A -85,B 0,C 180,E1 -24533.618,E2 -24533.618} C_VEL
LIN {X 0,Y 158.393,Z 535.893,A -85,B 0,C 180,E1 -24537.826,E2 -24537.826} C_VEL
LIN {X 0,Y 152.248,Z 534.871,A -85,B 0,C 180,E1 -24542.506,E2 -24542.506} C_VEL
LIN {X 0,Y 147.54,Z 532.718,A -85,B 0,C 180,E1 -24547.597,E2 -24547.597} C_VEL
LIN {X 0,Y 145.199,Z 530.555,A -85,B 0,C 180,E1 -24551.66,E2 -24551.66} C_VEL
LIN {X 0,Y 143.26,Z 533.531,A -85,B 0,C 180,E1 -24554.883,E2 -24554.883} C_VEL
LIN {X 0,Y 141.699,Z 535.17,A -85,B 0,C 180,E1 -24557.082,E2 -24557.082} C_VEL
LIN {X 0,Y 137.815,Z 537.192,A -85,B 0,C 180,E1 -24560.729,E2 -24560.729} C_VEL
LIN {X 0,Y 134.943,Z 538.228,A -85,B 0,C 180,E1 -24563.815,E2 -24563.815} C_VEL
LIN {X 0,Y 133.771,Z 538.754,A -85,B 0,C 180,E1 -24566.282,E2 -24566.282} C_VEL
LIN {X 0,Y 133.683,Z 538.88,A -85,B 0,C 180,E1 -24567.125,E2 -24567.125} C_VEL
LIN {X 0,Y 133.854,Z 539.084,A -85,B 0,C 180,E1 -24569.997,E2 -24569.997} C_VEL
LIN {X 0,Y 133.636,Z 538.84,A -85,B 0,C 180,E1 -24573.012,E2 -24573.012} C_VEL
LIN {X 0,Y 133.796,Z 537.163,A -85,B 0,C 180,E1 -24579.064,E2 -24579.064} C_VEL
LIN {X 0,Y 134.282,Z 535.702,A -85,B 0,C 180,E1 -24582.081,E2 -24582.081} C_VEL
LIN {X 0,Y 135.582,Z 532.686,A -85,B 0,C 180,E1 -24586.561,E2 -24586.561} C_VEL
LIN {X 0,Y 137.828,Z 528.621,A -85,B 0,C 180,E1 -24590.909,E2 -24590.909} C_VEL
LIN {X 0,Y 141.388,Z 522.366,A -85,B 0,C 180,E1 -24595.778,E2 -24595.778} C_VEL
LIN {X 0,Y 145.013,Z 515.546,A -85,B 0,C 180,E1 -24599.783,E2 -24599.783} C_VEL
LIN {X 0,Y 148.61,Z 508.592,A -85,B 0,C 180,E1 -24602.943,E2 -24602.943} C_VEL
LIN {X 0,Y 152.735,Z 500.209,A -85,B 0,C 180,E1 -24605.918,E2 -24605.918} C_VEL
LIN {X 0,Y 157.336,Z 489.844,A -85,B 0,C 180,E1 -24608.705,E2 -24608.705} C_VEL
LIN {X 0,Y 161.771,Z 478.184,A -85,B 0,C 180,E1 -24611.075,E2 -24611.075} C_VEL
LIN {X 0,Y 165.448,Z 466.449,A -85,B 0,C 180,E1 -24612.813,E2 -24612.813} C_VEL
LIN {X 0,Y 168.46,Z 454.312,A -85,B 0,C 180,E1 -24614.118,E2 -24614.118} C_VEL
LIN {X 0,Y 170.734,Z 441.9,A -85,B 0,C 180,E1 -24615.03,E2 -24615.03} C_VEL
LIN {X 0,Y 172.087,Z 428.064,A -85,B 0,C 180,E1 -24615.686,E2 -24615.686} C_VEL
LIN {X 0,Y 174.075,Z 397.004,A -85,B 0,C 180,E1 -24616.819,E2 -24616.819} C_VEL
LIN {X 0,Y 173.236,Z 382.57,A -85,B 0,C 180,E1 -24617.975,E2 -24617.975} C_VEL
LIN {X 0,Y 172.023,Z 379.738,A -85,B 0,C 180,E1 -24618.596,E2 -24618.596} C_VEL
LIN {X 0,Y 167.169,Z 370.94,A -85,B 0,C 180,E1 -24621.086,E2 -24621.086} C_VEL
LIN {X 0,Y 161.445,Z 361.564,A -85,B 0,C 180,E1 -24624.344,E2 -24624.344} C_VEL
LIN {X 0,Y 156.024,Z 353.67,A -85,B 0,C 180,E1 -24627.853,E2 -24627.853} C_VEL
LIN {X 0,Y 152.983,Z 349.533,A -85,B 0,C 180,E1 -24630.074,E2 -24630.074} C_VEL
LIN {X 0,Y 150.308,Z 345.921,A -85,B 0,C 180,E1 -24632.236,E2 -24632.236} C_VEL
LIN {X 0,Y 149.167,Z 344.722,A -85,B 0,C 180,E1 -24633.196,E2 -24633.196} C_VEL
LIN {X 0,Y 146.782,Z 341.833,A -85,B 0,C 180,E1 -24635.41,E2 -24635.41} C_VEL
LIN {X 0,Y 145.794,Z 340.087,A -85,B 0,C 180,E1 -24636.472,E2 -24636.472} C_VEL
LIN {X 0,Y 143.248,Z 338.061,A -85,B 0,C 180,E1 -24639.18,E2 -24639.18} C_VEL
LIN {X 0,Y 141.601,Z 334.957,A -85,B 0,C 180,E1 -24641.461,E2 -24641.461} C_VEL
LIN {X 0,Y 141.315,Z 334.414,A -85,B 0,C 180,E1 -24641.891,E2 -24641.891} C_VEL
LIN {X 0,Y 138.55,Z 332.84,A -85,B 0,C 180,E1 -24646.058,E2 -24646.058} C_VEL
LIN {X 0,Y 136.909,Z 330.154,A -85,B 0,C 180,E1 -24649.837,E2 -24649.837} C_VEL
LIN {X 0,Y 136.558,Z 328.42,A -85,B 0,C 180,E1 -24651.491,E2 -24651.491} C_VEL
LIN {X 0,Y 137.103,Z 328.404,A -85,B 0,C 180,E1 -24660,E2 -24660} C_VEL
LIN {X 0,Y 136.528,Z 328.517,A -85,B 0,C 180,E1 -24669.164,E2 -24669.164} C_VEL
LIN {X 0,Y 136.976,Z 330.362,A -85,B 0,C 180,E1 -24670.815,E2 -24670.815} C_VEL
LIN {X 0,Y 138.507,Z 332.862,A -85,B 0,C 180,E1 -24674.322,E2 -24674.322} C_VEL
LIN {X 0,Y 141.516,Z 334.639,A -85,B 0,C 180,E1 -24678.833,E2 -24678.833} C_VEL
LIN {X 0,Y 142.995,Z 337.72,A -85,B 0,C 180,E1 -24680.953,E2 -24680.953} C_VEL
LIN {X 0,Y 145.323,Z 339.826,A -85,B 0,C 180,E1 -24683.515,E2 -24683.515} C_VEL
LIN {X 0,Y 146.128,Z 340.516,A -85,B 0,C 180,E1 -24684.319,E2 -24684.319} C_VEL
LIN {X 0,Y 148.212,Z 343.81,A -85,B 0,C 180,E1 -24686.419,E2 -24686.419} C_VEL
LIN {X 0,Y 150.173,Z 345.724,A -85,B 0,C 180,E1 -24688.094,E2 -24688.094} C_VEL
LIN {X 0,Y 152.86,Z 349.439,A -85,B 0,C 180,E1 -24690.286,E2 -24690.286} C_VEL
LIN {X 0,Y 154.274,Z 351.366,A -85,B 0,C 180,E1 -24691.352,E2 -24691.352} C_VEL
LIN {X 0,Y 157.401,Z 355.696,A -85,B 0,C 180,E1 -24693.542,E2 -24693.542} C_VEL
LIN {X 0,Y 162.308,Z 362.967,A -85,B 0,C 180,E1 -24696.627,E2 -24696.627} C_VEL
LIN {X 0,Y 168.393,Z 373.02,A -85,B 0,C 180,E1 -24700.012,E2 -24700.012} C_VEL
LIN {X 0,Y 173.846,Z 383.435,A -85,B 0,C 180,E1 -24702.751,E2 -24702.751} C_VEL
LIN {X 0,Y 175.19,Z 386.272,A -85,B 0,C 180,E1 -24703.396,E2 -24703.396} C_VEL
LIN {X 0,Y 172.43,Z 425.509,A -85,B 0,C 180,E1 -24704.853,E2 -24704.853} C_VEL
LIN {X 0,Y 170.604,Z 438.77,A -85,B 0,C 180,E1 -24705.758,E2 -24705.758} C_VEL
LIN {X 0,Y 168.049,Z 451.064,A -85,B 0,C 180,E1 -24706.987,E2 -24706.987} C_VEL
LIN {X 0,Y 165.384,Z 461.279,A -85,B 0,C 180,E1 -24708.399,E2 -24708.399} C_VEL
LIN {X 0,Y 161.968,Z 471.646,A -85,B 0,C 180,E1 -24710.21,E2 -24710.21} C_VEL
LIN {X 0,Y 157.891,Z 482.254,A -85,B 0,C 180,E1 -24712.669,E2 -24712.669} C_VEL
LIN {X 0,Y 153.949,Z 491.495,A -85,B 0,C 180,E1 -24715.481,E2 -24715.481} C_VEL
LIN {X 0,Y 149.556,Z 500.289,A -85,B 0,C 180,E1 -24718.878,E2 -24718.878} C_VEL
LIN {X 0,Y 145.357,Z 507.746,A -85,B 0,C 180,E1 -24722.66,E2 -24722.66} C_VEL
LIN {X 0,Y 141.868,Z 513.723,A -85,B 0,C 180,E1 -24726.655,E2 -24726.655} C_VEL
LIN {X 0,Y 138.985,Z 518.442,A -85,B 0,C 180,E1 -24730.814,E2 -24730.814} C_VEL
LIN {X 0,Y 136.76,Z 522.044,A -85,B 0,C 180,E1 -24735.114,E2 -24735.114} C_VEL
LIN {X 0,Y 135.681,Z 523.894,A -85,B 0,C 180,E1 -24738.045,E2 -24738.045} C_VEL
LIN {X 0,Y 134.815,Z 525.304,A -85,B 0,C 180,E1 -24741.006,E2 -24741.006} C_VEL
LIN {X 0,Y 133.925,Z 526.898,A -85,B 0,C 180,E1 -24746.995,E2 -24746.995} C_VEL
LIN {X 0,Y 133.848,Z 527.125,A -85,B 0,C 180,E1 -24750.003,E2 -24750.003} C_VEL
LIN {X 0,Y 134.191,Z 526.428,A -85,B 0,C 180,E1 -24755.679,E2 -24755.679} C_VEL
LIN {X 0,Y 134.798,Z 525.374,A -85,B 0,C 180,E1 -24759.002,E2 -24759.002} C_VEL
LIN {X 0,Y 135.647,Z 524.005,A -85,B 0,C 180,E1 -24761.964,E2 -24761.964} C_VEL
LIN {X 0,Y 137.357,Z 521.131,A -85,B 0,C 180,E1 -24766.348,E2 -24766.348} C_VEL
LIN {X 0,Y 139.817,Z 517.214,A -85,B 0,C 180,E1 -24770.604,E2 -24770.604} C_VEL
LIN {X 0,Y 142.894,Z 512.138,A -85,B 0,C 180,E1 -24774.715,E2 -24774.715} C_VEL
LIN {X 0,Y 146.605,Z 505.735,A -85,B 0,C 180,E1 -24778.648,E2 -24778.648} C_VEL
LIN {X 0,Y 151.053,Z 497.751,A -85,B 0,C 180,E1 -24782.351,E2 -24782.351} C_VEL
LIN {X 0,Y 155.03,Z 489.24,A -85,B 0,C 180,E1 -24785.469,E2 -24785.469} C_VEL
LIN {X 0,Y 159.154,Z 479.516,A -85,B 0,C 180,E1 -24788.189,E2 -24788.189} C_VEL
LIN {X 0,Y 162.907,Z 469.558,A -85,B 0,C 180,E1 -24790.328,E2 -24790.328} C_VEL
LIN {X 0,Y 166.286,Z 458.703,A -85,B 0,C 180,E1 -24792.143,E2 -24792.143} C_VEL
LIN {X 0,Y 169.279,Z 446.623,A -85,B 0,C 180,E1 -24793.651,E2 -24793.651} C_VEL
LIN {X 0,Y 171.623,Z 433.423,A -85,B 0,C 180,E1 -24794.806,E2 -24794.806} C_VEL
LIN {X 0,Y 173.124,Z 420.455,A -85,B 0,C 180,E1 -24795.509,E2 -24795.509} C_VEL
LIN {X 0,Y 175.34,Z 386.353,A -85,B 0,C 180,E1 -24796.758,E2 -24796.758} C_VEL
LIN {X 0,Y 169.569,Z 374.9,A -85,B 0,C 180,E1 -24799.619,E2 -24799.619} C_VEL
LIN {X 0,Y 163.535,Z 364.722,A -85,B 0,C 180,E1 -24802.915,E2 -24802.915} C_VEL
LIN {X 0,Y 158.527,Z 357.239,A -85,B 0,C 180,E1 -24805.99,E2 -24805.99} C_VEL
LIN {X 0,Y 155.847,Z 353.428,A -85,B 0,C 180,E1 -24807.812,E2 -24807.812} C_VEL
LIN {X 0,Y 154.059,Z 350.865,A -85,B 0,C 180,E1 -24809.122,E2 -24809.122} C_VEL
LIN {X 0,Y 153.622,Z 350.765,A -85,B 0,C 180,E1 -24809.406,E2 -24809.406} C_VEL
LIN {X 0,Y 151.646,Z 353.9,A -85,B 0,C 180,E1 -24810.405,E2 -24810.405} C_VEL
LIN {X 0,Y 149.441,Z 355.742,A -85,B 0,C 180,E1 -24811.756,E2 -24811.756} C_VEL
LIN {X 0,Y 146.066,Z 367.245,A -85,B 0,C 180,E1 -24813.09,E2 -24813.09} C_VEL
LIN {X 0,Y 143.876,Z 373.335,A -85,B 0,C 180,E1 -24814.179,E2 -24814.179} C_VEL
LIN {X 0,Y 142.592,Z 375.63,A -85,B 0,C 180,E1 -24815.005,E2 -24815.005} C_VEL
LIN {X 0,Y 142.035,Z 375.372,A -85,B 0,C 180,E1 -24815.526,E2 -24815.526} C_VEL
LIN {X 0,Y 141.858,Z 373.291,A -85,B 0,C 180,E1 -24815.94,E2 -24815.94} C_VEL
LIN {X 0,Y 141.874,Z 371.812,A -85,B 0,C 180,E1 -24816.121,E2 -24816.121} C_VEL
LIN {X 0,Y 139.68,Z 424.884,A -85,B 0,C 180,E1 -24821.576,E2 -24821.576} C_VEL
LIN {X 0,Y 138.837,Z 439.437,A -85,B 0,C 180,E1 -24823.647,E2 -24823.647} C_VEL
LIN {X 0,Y 138.044,Z 452.268,A -85,B 0,C 180,E1 -24826.055,E2 -24826.055} C_VEL
LIN {X 0,Y 137.114,Z 465.61,A -85,B 0,C 180,E1 -24829.292,E2 -24829.292} C_VEL
LIN {X 0,Y 136.504,Z 476.545,A -85,B 0,C 180,E1 -24832.605,E2 -24832.605} C_VEL
LIN {X 0,Y 136.059,Z 486.514,A -85,B 0,C 180,E1 -24836.298,E2 -24836.298} C_VEL
LIN {X 0,Y 135.89,Z 494.798,A -85,B 0,C 180,E1 -24840,E2 -24840} C_VEL
LIN {X 0,Y 135.817,Z 502.946,A -85,B 0,C 180,E1 -24844.452,E2 -24844.452} C_VEL
LIN {X 0,Y 136.252,Z 509.675,A -85,B 0,C 180,E1 -24848.902,E2 -24848.902} C_VEL
